(* CoDeSys 2.3 project: cy-08-wg-03.pro *)
(* Title: ClevergyAS - SanFelice *)
(* Version: 0.0 *)
(* Author: Andrea Ravasio *)
(* Libraries: serial_interface_01.lib 22.4.13 12:50:14, SerComm.lib 31.5.11 08:54:36, MBus_03.lib 9.2.13 17:51:58, Util.lib 18.5.10 15:14:28, Visual.lib 2.12.10 14:48:34, WagoLibIdent.lib 25.2.13 11:12:16, WagoLibStatus.lib 2.12.10 14:48:32, SysLibFile.lib 2.12.10 14:48:34, SysLibRtc.lib 2.12.10 14:48:32, SysLibSockets.lib 10.2.11 09:20:54, SysLibEvent.lib 2.12.10 14:48:34, SysLibPlcCtrl.lib 2.12.10 14:48:32, Standard.lib 2.12.10 14:48:34, SYSLIBCALLBACK.LIB 2.12.10 14:48:32, WagoLibModbus_IP_01.lib*24.7.13 15:05:58 *)

(* PLC configuration (modules and I/O channels)
0750-0402 4 DI 24 V DC 3.0ms [Type_1_4_Channels] node 0, in %IB0 out %QB0 {INTTypePAAssignment = PLC; INTTypeModule = plugged}
  AT %IX0.0 [BOOLOnX_I] Ch_1 Digital input
  AT %IX0.1 [BOOLOnX_I] Ch_2 Digital input
  AT %IX0.2 [BOOLOnX_I] Ch_3 Digital input
  AT %IX0.3 [BOOLOnX_I] Ch_4 Digital input
Fieldbus variables [FB_VARS] node 1, in %IB0 out %QB0
Flag variables [FLAG_VARS] node 2, in %IB0 out %QB0
Modbus-Master [MB_MASTER] node 3, in %IB0 out %QB0
*)

(* Global variable list: Global_Constants *)
VAR_GLOBAL CONSTANT

	Plant_SN			: DWORD :=8;   		(* S/N Impianto di telecontrollo *)
	Plant_SW_VER		: WORD  :=3;		(* Versione SW installata *)

	(* Parameters *)

	(* Filesystem *)
	FilesPath  			: STRING :='S:\';

	(* TCP Logger *)
	Logger_SERVER			: STRING:='';
	Logger_IP					: STRING:='178.33.227.41'; (*192.168.100.3'; (*' clevergyimpianti.it  *)*)
	Logger_PORT				: WORD  :=80;
	Logger_GETSTART		: STRING:='GET /cygmsrv/hsgm.ashx?';
	Logger_GETEND			: STRING:='$R$N$R$N';
	Logger_CHECK			: STRING:='True';
	Logger_CRLF				: STRING:='$R$N';
	Logger_DataFile			: STRING:='S:\LOG.DAT';
	Logger_DataFileOld		: STRING:='S:\LOG.BCK';
	Logger_IndexFile			: STRING:='S:\LOG.IDX';
	Logger_ConnRetries		: BYTE:=5;
	Logger_RecoverMsgs	: BYTE:=100;

	(* TCP Remote *)
	Remote_PORT			: WORD  :=44818;
	Remote_WELCOME		: STRING:='Connected$R$N';
	Remote_OK				: STRING:='OK$R$N';
	Remote_ERROR			: STRING:='ERROR$R$N';

	(* TCP Sockets *)
	MAX_SEND_TCP_SERVER					 : DWORD:=3000;(*60000*)
	MAX_RECEIVE_TCP_SERVER				 : DWORD:=3000;
	MAX_RECEIVE_TCP_SERVER_SOCKET	  : DWORD:=1500;
	MAX_SEND_TCP_CLIENT					 : DWORD:=3000;(*15000*)
	MAX_RECEIVE_TCP_CLIENT				 : DWORD:=1500;
	MAX_RECEIVE_TCP_CLIENT_SOCKET		 : DWORD:=1500;
	MAX_RECEIVE_UDP_SERVER				 : INT  :=1472;
	MAX_RECEIVE_UDP_CLIENT				 : INT  :=1472;
	CONNECT_WATCHDOG_TIME				 : TIME :=t#10s;

END_VAR

VAR_GLOBAL CONSTANT RETAIN
	TiemOutModbus_TCPIP				: TIME:=t#40ms;
	OffsetIndirizzo				: WORD := 0;(*12288;    (* questo servere per leggere il nodo WAGO *) *)

	MaxRigheFileCSV			:BYTE:=30; (* Massimo riche da leggere del afile csv *)
	MAXCaratteri				:WORD:=6000; (*Numero Massimo di caratteri da leggere dal file equivale alla lunghezza dei file*)


END_VAR

(* Global variable list: Global_Retain *)
VAR_GLOBAL RETAIN PERSISTENT
(*	CTL01_Count : DWORD;

	PortataTotalePORT01: DINT;
	ConteggioTotalePORT01: DINT;
	PortataTotaleGAS01: DINT;
	ConteggioTotaleGAS01: DINT;
	PortataTotaleGAS02: DINT;
	ConteggioTotaleGAS02: DINT;
*)
	Mode_Manual : BOOL := FALSE;
END_VAR

(* Global variable list: Global_Variables *)
VAR_GLOBAL

	SYS    : typ_SYS;


(* PLC *)

	Sistem_Status 							: INT ;
	BATTERY_STATUS 						: INT ;
	SYSTEM_STATUS_COMMAND 			: WORD;
	STATUS_DIGITAL_INPUT_1 				: WORD;
	STATUS_DIGITAL_OUTPUT_1			: WORD;
	STATUS_SYSTEM_WARNNG_1  			: WORD;
	STATUS_SYSTEM_ALARM_1 			: WORD;
	STATUS_SYSTEM_ALARM_2 			: WORD;

	PM1_Voltage_L12 						:REAL;
	PM1_Voltage_L23							:REAL;
	PM1_Voltage_L31 						:REAL;
	PM1_Current_L12						:REAL;
	PM1_Current_L23 						:REAL;
	PM1_Current_L31 						:REAL;
	PM1_Active_Power_Total 				:REAL;
	PM1_Reactive_Power_Total				:REAL;
	PM1_Apparent_Power_Total 				:REAL;
	PM1_Frequency 							:REAL;
	PM1_Power_Factor_Total 				:REAL;

(* GATEWAY BATTERY*)

	GW_Actual_DC_Voltage 					:REAL;
	GW_Actual_DC_Current 					:REAL;
	GW_Actual_Battery_SOC 				:REAL;
	GW_Actual_Heaters_Current 			:REAL;
	GW_Vdc_Link_Request 					:REAL;
	GW_Limit_Discharge_Current 			:REAL;
	GW_Limit_Charge_Current 				:REAL;
	GW_Min_DC_Voltage 					:REAL;
	GW_Max_DC_Voltage					:REAL;
	GW_Actual_Battery_Capacity 			:REAL;
	GW_Max_Battery_Voltage 				:REAL;
	GW_Min_Battery_Voltage 				:REAL;
	GW_Max_Battery_Temperature			:REAL;
	GW_Min_Battery_Temperature 			:REAL;
	GW_Actual_DC_Power 					:REAL;
	GW_HOURSOp_Time  					:INT;
	GW_MINOp_Time 						:INT;
	GW_Status_Warning_1 					:INT;
	GW_Status_Warning_2 					:INT;
	GW_Status_Alarm_1 						:INT;
	GW_Status_Alarm_2 						:INT;
	GW_Status_Warning_A 					:INT;
	GW_Status_Warning_B 					:INT;
	GW_Status_Alarm_A 						:INT;
	GW_CONTROLWORD  					:WORD ;
	GW_STATUSWORD  						:WORD;



(* PCS HPP 35*)

	PCS_Actual_Current_R 					 :REAL;
	PCS_Actual_Current_S 					 :REAL;
	PCS_Actual_Current_T 					 :REAL;
	PCS_Actual_Voltage_RS					 :REAL;
	PCS_Actual_Voltage_ST 					 :REAL;
	PCS_Actual_Voltage_TR					 :REAL;
	PCS_Frequency 							 :REAL;
	PCS_P_Actual 							 :REAL;
	PCS_Q_Actual 							 :REAL;
	PCS_A_Actual 							 :REAL;
	PCS_Battery_Voltage 						 :REAL;
	PCS_Battery_Current						 :REAL;
	PCS_Battery_Power 						 :REAL;
	PCS_PV_Voltage 							 :REAL;
	PCS_PV_Current 							 :REAL;
	PCS_PV_Power							 :REAL;
	PCS_HPP_Status 						 :INT;
	PCS_Drive_Status 						 :INT;
	PCS_Chopper_Status 					 :INT;
	PCS_Run_Mode 							 :INT;
	PCS_Drive_Warning_1  					 :WORD;
	PCS_Drive_Alarm_1  						 :WORD;
	PCS_HPP_Warning_1  					 :WORD;
	PCS_HPP_Alarm_1 						 :WORD ;


(* Write Register*)

	Ref_P										:REAL;

(* Variabile letta dal file CSV *)

	Ref_AvctivePower							:REAL;
	NomeFileSchedulazione					:STRING:='S:\Schedulazione.csv' ;
	WebStrutturaDati							: ARRAY [1..MaxRigheFileCSV] OF StrutturaDatiCSV;
	ForzaLetturaCSV: BOOL;

(* Variabile lettura ModBus ETH *)

	BitConnessione: BOOL ;    (* Abilita Comunicazione ModBus TCP-IP *)
	StartComunicazione: BOOL;
	ForzaLettura: BOOL;


	Logger : typ_Logger;

	(**** SIMULATION ONLY ****)
	TEST1		:BOOL;
	TEST2		:BOOL;

	T_S1		:INT:=100;

END_VAR


VAR_GLOBAL CONSTANT

END_VAR

(* Data type in Errors *)
TYPE en_Logger_ErrLev :
(
	EL_Log			:=0,
	EL_Wrn			:=1,
	EL_Alarm		:=2,
	EL_AlarmStop	:=3
);
END_TYPE

(* Data type in Errors *)
TYPE en_Logger_Status :
(
	S_Logger_UNKNOWN := 0,
	S_Logger_IDLE,
	S_Logger_WAITCONN,
	S_Logger_WAITTX,
	S_Logger_WAITRESP,
	S_Logger_ERROR
);
END_TYPE

(* Data type *)
TYPE en_SYS_Objects :
(
	EO_SYS		:=0,  (* PLC *)
	EO_VPN		:=1,  (* VPN *)
	EO_DOOR		:=2,  (* Door & access control *)

	EO_CAL		:=10, (* Caldaia *)
	EO_CIR		:=11, (* Circolatore *)
	EO_CRON		:=12, (* Crono-termostato *)
	EO_VRD		:=13, (* Valvola miscelatore pannelli *)
	EO_CTL		:=14, (* Contalitri *)
	EO_CTB		:=15, (* Contabilizzatore *)
	EO_TPV		:=16, (* Temperature probes & values *)
	EO_PPV		:=17, (* Pressure probes & values *)
	EO_PBV		:=18, (* Over-Pressure Alarms *)
	EO_TBV		:=19, (* Over-Temperature Alarms *)
	EO_PMV		:=20, (* Under-Pressure Alarms *)
	EO_GRU		:=21, (* Gruppo termico *)
	EO_PDC		:=22, (* Pompa di calore *)
	EO_SOL		:=23, (* Pannello solare termico *)
	EO_ESOL		:=24, (* Pannello solare fotovoltaico *)
	EO_GAS		:=25, (* Contatore GAS *)
	EO_PORT		:=26, (* Misuratore di portata *)

	EO_LON		:=1000, (* Bus - LON *)
	EO_MODBUS	:=1001, (* Bus - MODBUS *)
	EO_MBUS		:=1002  (* Bus - M-BUS *)
);
END_TYPE

(* Data type *)
TYPE en_SYS_Status :
(
	S_UNKNOWN  := 0,
	S_STARTUP,
	S_INIT_RTC,
	S_INIT_VAR,
	S_AUTOTEST,
	S_RUNNING,
	S_SHUTDOWN,
	S_HALT
);
END_TYPE

(* Data type in Plant_Objects *)
TYPE StrutturaDatiCSV :

STRUCT

	sdIndice: STRING(3);
	sdData: STRING(12);
	sdOra: STRING(6);
	sdOrigine: STRING(12);
	sdVaribile: STRING(10);
	sdValore: STRING(10);
END_STRUCT
END_TYPE

(* Data type in Plant_Objects *)
TYPE Typ_CTB_MBUS :
STRUCT
	Value			: STRING[21];
	Pof10			: STRING[3];
	Unit			: STRING[7];
	Descriptor		: STRING[6];
	(*Enum_Unit	: typMBusUnit; *)
END_STRUCT
END_TYPE

(* Data type in Errors *)
TYPE typ_Logger :
STRUCT
	Status		: en_Logger_Status;

	SendReq		: BOOL;
	SendIdx		: DWORD;
	SendData	: ARRAY [0..MAX_SEND_TCP_CLIENT] OF BYTE;
	SendLen		: DINT;

	TData		: ARRAY [0..MAX_SEND_TCP_CLIENT] OF BYTE;
	TLen		: DINT;

	LastIdxPos	: DWORD;

END_STRUCT
END_TYPE

(* Data type *)
TYPE typ_SYS :
STRUCT
	Status			: en_SYS_Status;
	Warning			: BOOL;
	Alarm			: BOOL;
	AlarmStop		: BOOL;

	Time_LogString	: STRING;
	Time_Year		: WORD;
	Time_Month		: BYTE;
	Time_Day		: BYTE;

	Time_CT_DT		: DT;
	Time_CT_Day		: WORD;
	Time_CT_Quarter	: BYTE;

	LastLogs_Idx	: BYTE;
	LastLogs_Dat	: ARRAY[0..5] OF STRING;
	LastLogs_Msg	: ARRAY[0..5] OF STRING;

END_STRUCT
END_TYPE

(* Data type in Plant_Objects *)
TYPE typ_VisuStrutturaMbus :
STRUCT

	sdNodoPresente: STRING(16);
	sdEnergia: STRING(16);
	sdPotenza: STRING(16);
	sdVolume: STRING(16);
	sdFlow: STRING(16);
	sdTempIngresso: STRING(8);
	sdTempaUscita: STRING(8);
	sdTempDelta: STRING(8);

END_STRUCT
END_TYPE

(* POU PLC_PRG, ST *)
PROGRAM PLC_PRG
VAR
	Timer1: TON; (* Fast controls tick *)
	Timer2: TON; (* Plant control tick *)
	Timer3: TON; (* Logger timer *)
	Timer4: TON; (* Logger timer *)
END_VAR
(******************************************************************************
 ****                           MAIN TASK CODE                             ****
 ******************************************************************************

	Network setup:
		IP  = 10.186.73.101 | MSK = 255.255.255.0 | GW = 10.186.73.254 
		DNS = ___.___.___.___ | NTP = ___.___.___.___

	Editor setup:
		Project --> Options --> Editor --> Fonts --> Courier NEW / BOLD / 12

*)

(*==============================*)
(*===== Main status machine ====*)
(*==============================*)
Main_Stm();
SceltaWrite();
(*=====================================*)
(*== Running common cycle operations ==*)
(*=====================================*)

IF SYS.Status>S_INIT_VAR THEN

(*	(* Execute M-BUS processes *)
	MBUS01();
	CTBSCAN01( MBus:=MBUS01.MBus ); *)

	ModBus_TCPIP();



END_IF

(*==============================*)
(*== System cycle operations ===*)
(*==============================*)
(* Execute TCP processes *)
Logger_Proc();
Remote_Proc();
(* Update user led *)
USRLED_Update();
(* Execute Cron Editor commands *)
(*...*)
(* External resources *)
(*...*)

(**** SIMULATION ONLY ****)
(*...*)
END_PROGRAM
ACTION Main_Stm:
CASE Sys.Status OF

	S_STARTUP:
		Sys.Status:=S_INIT_RTC;
		BitConnessione:=FALSE;

	S_INIT_RTC:
		(* Check RTC and update from network *)
		RTC_Update();
		(* Check time *)
		IF Sys.Time_Year>2000 THEN
			Sys.Status:=S_INIT_VAR;
		END_IF

	S_INIT_VAR:
		LogEv(EL_Wrn,EO_SYS,0,1,CONCAT('System_startup_v',WORD_TO_STRING(Plant_SW_VER)));
		Sys.Status:=S_RUNNING;
		BitConnessione:=TRUE;
		PRG_ApriFile( NomeFile:=NomeFileSchedulazione  ,  LungRecord:=4 );

	S_RUNNING:

		Timer1(IN:=NOT Timer1.Q,PT:=T#50ms);
(*		IF Timer1.Q THEN
			(* Update system checks *)
			(*SYS_Proc();*)
		END_IF
*)

		Timer2(IN:=NOT Timer2.Q AND NOT ForzaLettura ,PT:=T#10s); (* Lettura Variabili PLC Siemens via TCP-IP *)
		IF Timer2.Q OR ForzaLettura THEN
			(* Read current date/time *)
			RTC_Update();
			(* === Execute plant operations === *)
			StartComunicazione:=TRUE;
			(* Test toggle *)
			IF TEST1 THEN TEST1:=FALSE; ELSE TEST1:=TRUE; END_IF
		     END_IF

		Timer3(IN:=NOT Timer3.Q,PT:=T#5m);
		IF Timer3.Q THEN
			(* Trig logger *)
			LogTrig();
			(* Execute temporary CSV logger *)
(*			CSV_Log(); *)
		END_IF

		Timer4(IN:=NOT Timer4.Q AND NOT ForzaLetturaCSV,PT:=T#5m);    (* Lettura File Struttura *)
		IF Timer4.Q OR ForzaLetturaCSV THEN
			PRG_ApriFile( NomeFile:=NomeFileSchedulazione  ,  LungRecord:=4 );
		END_IF





	S_SHUTDOWN:
		(* Arresto del sistema *)
		Sys.Status:=S_STARTUP;
		BitConnessione:=FALSE;
	S_HALT:
		(* Aspetta uscita manuale *)
		Sys.Status:=S_STARTUP;


ELSE
	Sys.Status:=S_STARTUP;
END_CASE;
END_ACTION

(* POU Utils/SceltaWrite, ST *)
PROGRAM SceltaWrite
VAR
	TS: STRING;
	ORAttuale: INT;

	x: INT;
	OraImpostata: INT;
	StringaAggiornata: BOOL;
	Ref_AvctivePowerold: REAL;
END_VAR
(* scelgo la varibile da scrivere in funzione del'ora *)




(* Calculate variables *)
TS:=DT_TO_STRING(Sys.Time_CT_DT);
ORAttuale:=STRING_TO_INT(MID(STR:=TS, LEN:=2, POS:=15));


FOR x:=1 TO PRG_ApriFile.Riga BY 1 DO
       OraImpostata :=STRING_TO_INT(LEFT(WebStrutturaDati[x].sdOra,2));
	IF ORAttuale>=OraImpostata THEN
		Ref_AvctivePower:=STRING_TO_REAL((WebStrutturaDati[x].sdValore ));
		END_IF
END_FOR

IF Ref_AvctivePower <>  Ref_AvctivePowerold THEN
		 LogEv(EL_Log,0,3,1,'Reference_active_power_Aggiornato');    (*********************************** moreno **********************)
		 Ref_AvctivePowerold:=Ref_AvctivePower;
END_IF
END_PROGRAM

(* POU Utils/PRG_ApriFile, ST *)
PROGRAM PRG_ApriFile


VAR
	(* Varibili per l'apertura del del File CVS *)
	xStart:							BOOL;

	FileIdent: 						DWORD;
	CarattereLetto:				ARRAY[0..50000] OF BYTE;
	filesizev: 						DINT;
(*	RecordLetto: 					STRING(80); *)
	PrimoCarattereRiga: 			INT;
	NumCaratteri:					DINT;
	Record: 						INT;
	Carattere: 						STRING(1);

	Riga: INT;
(*	x: DWORD;*)

	StringaAppoggio: STRING;
	Valore2: REAL;

(*	BufferLetto:			ARRAY[0..186] OF BYTE; *)


	NumeroRighe: BOOL;
(*	bCarattere: BYTE; *)
	AggiornaDato: BOOL;

END_VAR

VAR_INPUT
	NomeFile:STRING(20);
	LungRecord: BYTE;
END_VAR
(* cerco il file se presente quindi dò l'OK*)


	FileIdent:=SysFileOpen(FileName:=NomeFile , Mode:='r');
	IF fileident<>0 THEN
		SysFileRead(File:=Fileident, Buffer:=ADR(CarattereLetto), Size:=SIZEOF(CarattereLetto));
		filesizev:=SysFileGetSize(FileName:=NomeFile);
		NumeroRighe:=SysFileEOF(FileIdent);
		IF filesizev>MAXCaratteri THEN
			filesizev:=MAXCaratteri;
		END_IF
		SysFileClose(File:=fileident);(*this function is blocking*)
		xStart:=TRUE;
	ELSE
		xStart:=FALSE;
		LogEv(EL_Alarm,0,3,1,'Errore_File_CSV_Non_Letto');    (*********************************** moreno **********************)

		RETURN;(*no such file available*)
	END_IF

IF xStart=TRUE THEN



	PrimoCarattereRiga:=0;
	NumCaratteri:=0;
	Record:=1;
	Riga:=1;
	StringaAppoggio:='';

(* Costruisco la stringa *)

		FOR NumCaratteri:=0 TO filesizev DO

					(* elimino i caratteri che non mi servono *)

					WHILE  CarattereLetto[NumCaratteri]=10 OR (*Caratterre ? *)
						(*	 CarattereLetto[NumCaratteri]=32 OR (*Caratterre   *) *)
							 CarattereLetto[NumCaratteri]=34 OR (*Caratterre " *)
							 CarattereLetto[NumCaratteri]=36 OR (*Caratterre ' *)
							 CarattereLetto[NumCaratteri]=39 DO
 							NumCaratteri:=NumCaratteri+1;
					END_WHILE


					(* Gestione Caratteri di controllo *)
					IF CarattereLetto[NumCaratteri]=13 THEN  (*Caratterre fine Riga  *)
						AggiornaDato:=TRUE;
					 END_IF
					IF CarattereLetto[NumCaratteri]=59 THEN (*Caratterre Separatore Record*)
						AggiornaDato:=TRUE;
					 END_IF

			IF aggiornaDato THEN

					(*Creo l'array nel PLC dei valori letti dal file  *)
				CASE Record OF

						1:	WebStrutturaDati[Riga].sdIndice:=INT_TO_STRING(RIGA);
							WebStrutturaDati[Riga].sdData:=LEFT(StringaAppoggio,10);
							WebStrutturaDati[Riga].sdOra:=RIGHT(StringaAppoggio,5);
							Record:=Record+1;
						2: 	WebStrutturaDati[Riga].sdOrigine:=StringaAppoggio;
							Record:=Record+1;
						3: 	WebStrutturaDati[Riga].sdVaribile:=StringaAppoggio;
							Record:=Record+1;
						4: 	WebStrutturaDati[Riga].sdValore:=StringaAppoggio;
							Record:=Record+1;

				END_CASE
				AggiornaDato:=FALSE;
				StringaAppoggio:='';
				IF Record>LungRecord THEN
						Record:=1;
						Riga:=Riga+1;
				 END_IF



			ELSE
					Carattere:=FUN_ByteAsci(CarattereLetto[NumCaratteri]);
					StringaAppoggio:=CONCAT(StringaAppoggio,Carattere);
			END_IF
		END_FOR

END_IF
END_PROGRAM

(* POU TCP_Logger/LogEv, ST *)
FUNCTION LogEv : BOOL
VAR_INPUT
	Level	: en_Logger_ErrLev;
	Object  : en_SYS_Objects;
	Index	: WORD;
	Error	: WORD;
	Message : STRING;
END_VAR
VAR
	s1 : STRING(160);
	i  : INT;
END_VAR
(* Execute error level operations *)
CASE Level OF
	EL_Wrn: 	Sys.Warning:=TRUE;
	EL_Alarm: 		Sys.Alarm:=TRUE;
	EL_AlarmStop: 	Sys.Alarm:=TRUE; (* GO TO STOP STATE!! *)
END_CASE

(* Fill lastlog list *)
s1:=CONCAT(Sys.Time_LogString,';Lev=');
s1:=CONCAT(s1,INT_TO_STRING(Level));
s1:=CONCAT(s1,';Obj=');
s1:=CONCAT(s1,INT_TO_STRING(Object));
s1:=CONCAT(s1,';Idx=');
s1:=CONCAT(s1,WORD_TO_STRING(Index));
s1:=CONCAT(s1,';Err=');
s1:=CONCAT(s1,WORD_TO_STRING(Error));
Sys.LastLogs_Dat[Sys.LastLogs_Idx]:=s1;
Sys.LastLogs_Msg[Sys.LastLogs_Idx]:=Message;
Sys.LastLogs_Idx:=Sys.LastLogs_Idx+1;
IF Sys.LastLogs_Idx>5 THEN Sys.LastLogs_Idx:=0; END_IF

(*---------------------------------------------------------------*)
(*---------------------------------------------------------------*)
Logger.TLen:=0;
(* Set GET header *)
ADDSTRING(ADR(Logger.TData), ADR(Logger_GETSTART), Logger.TLen);

(* Insert Header *)
s1:=INSERT('ID=&V=1&D=',DWORD_TO_STRING(Plant_SN),3);
s1:=CONCAT(s1,Sys.Time_LogString);
s1:=CONCAT(s1,'&S=');
IF Sys.Alarm THEN i:=2; ELSIF Sys.Warning THEN i:=1; ELSE i:=0; END_IF
s1:=CONCAT(s1,INT_TO_STRING(i));
ADDSTRING(ADR(Logger.TData), ADR(s1), Logger.TLen);

(* Insert ERR *)
s1:=CONCAT('&ERR=',INT_TO_STRING(Level));
s1:=CONCAT(s1,';');
s1:=CONCAT(s1,INT_TO_STRING(Object));
s1:=CONCAT(s1,';');
s1:=CONCAT(s1,WORD_TO_STRING(Index));
s1:=CONCAT(s1,';');
s1:=CONCAT(s1,WORD_TO_STRING(Error));
s1:=CONCAT(s1,';');
ADDSTRING(ADR(Logger.TData), ADR(s1), Logger.TLen);
s1:=Message;
ADDSTRING(ADR(Logger.TData), ADR(s1), Logger.TLen);

(* Finalize string *)
ADDSTRING(ADR(Logger.TData), ADR(Logger_GETEND), Logger.TLen);

(*---------------------------------------------------------------*)
(*---------------------------------------------------------------*)

Logger_Send();
END_FUNCTION

(* POU Utils Functions/ADDSTRING, ST *)
FUNCTION ADDSTRING : BOOL
VAR_INPUT
	pTxData: POINTER TO BYTE;
	pString: POINTER TO BYTE;
END_VAR
VAR_IN_OUT
	TxLen: DINT;
END_VAR
VAR
END_VAR
pTxData:=pTxData+TxLen;
WHILE pString^<>0 DO
	pTxData^:=pString^;
	pString:=pString+1;
	pTxData:=pTxData+1;
	TxLen:=TxLen+1;
END_WHILE
END_FUNCTION

(* POU TCP_Logger/Logger_Send, ST *)
FUNCTION Logger_Send : BOOL
VAR
	hFile: 	DWORD;
	pos:	DWORD;
END_VAR
(* Read log position *)
pos:=SysFileGetSize(Logger_DataFile);
(* Check log size, bckup and erase if no pending messages *)
IF pos>100000000 (*100M*) THEN
	hFile:=SysFileOpen(Logger_IndexFile,'r');
	IF hFile=0 THEN
		SysFileDelete(Logger_DataFileOld);
		SysFileRename(Logger_DataFile,Logger_DataFileOld);
		pos:=0;
	ELSE
		SysFileClose(hFile);
	END_IF
END_IF
(* Write message on log file *)
hFile:=SysFileOpen(Logger_DataFile,'a');
IF hFile<>0 THEN
	SysFileWrite(hFile, ADR(Logger.TData), Logger.TLen);
	SysFileClose(hFile);
ELSE
	Sys.Warning:=TRUE;
END_IF


(* Check logger status *)
IF Logger.SendReq=FALSE THEN
	(* Set log position for recovery *)
	Logger.SendIdx:=pos;
	(* Copy message data *)
	MEMCPY(ADR(Logger.TData),ADR(Logger.SendData),DINT_TO_WORD(Logger.TLen));
	Logger.SendLen:=Logger.TLen;
	(* Trigger request *)
	Logger.SendReq:=TRUE;
ELSE
	(* Add message position+size in recovery indexes *)
	hFile:=SysFileOpen(Logger_IndexFile,'a');
	SysFileWrite(hFile, ADR(pos), SIZEOF(pos));
	SysFileWrite(hFile, ADR(Logger.TLen), SIZEOF(Logger.TLen));
	SysFileClose(hFile);
END_IF
END_FUNCTION

(* POU Utils Functions/MEMCPY, ST *)
FUNCTION MEMCPY:BOOL
VAR_INPUT
	pSourceAddress:POINTER TO ARRAY[1..2] OF BYTE;
	pDestinationAddress:POINTER TO ARRAY[1..2] OF BYTE;
	BytesToCopy:WORD;
END_VAR
VAR
END_VAR
WHILE (BytesToCopy > 0) DO
	pDestinationAddress^[1]:=pSourceAddress^[1]; (* copy bytes from source to destination *)
	pDestinationAddress:=ADR(pDestinationAddress^[2]); (* increment destination *)
	pSourceAddress:=ADR(pSourceAddress^[2]);(* increment source *)
	BytesToCopy:=BytesToCopy -1; (* decrement number of bytes to copy *)
END_WHILE
END_FUNCTION

(* POU IMI/FUN/FUN_ByteAsci, ST *)
FUNCTION FUN_ByteAsci : STRING(1)
VAR_INPUT
	ByteIn:BYTE;
END_VAR
VAR
END_VAR
CASE ByteIn OF

	32: FUN_ByteAsci:=' ';
	33: FUN_ByteAsci:='!';
	34: FUN_ByteAsci:='"';
	35: FUN_ByteAsci:='#';

	37: FUN_ByteAsci:='%';
	38: FUN_ByteAsci:='&';

	40: FUN_ByteAsci:='(';
	41: FUN_ByteAsci:=')';
	42: FUN_ByteAsci:='*';
	43: FUN_ByteAsci:='+';
	44: FUN_ByteAsci:=',';
	45: FUN_ByteAsci:='-';
	46: FUN_ByteAsci:='.';
	47: FUN_ByteAsci:='/';
	48: FUN_ByteAsci:='0';
	49: FUN_ByteAsci:='1';
	50: FUN_ByteAsci:='2';
	51: FUN_ByteAsci:='3';
	52: FUN_ByteAsci:='4';
	53: FUN_ByteAsci:='5';
	54: FUN_ByteAsci:='6';
	55: FUN_ByteAsci:='7';
	56: FUN_ByteAsci:='8';
	57: FUN_ByteAsci:='9';
	58: FUN_ByteAsci:=':';
	59: FUN_ByteAsci:=';';
	60: FUN_ByteAsci:='<';
	61: FUN_ByteAsci:='=';
	62: FUN_ByteAsci:='>';
	63: FUN_ByteAsci:='?';
	64: FUN_ByteAsci:='@';
	65: FUN_ByteAsci:='A';
	66: FUN_ByteAsci:='B';
	67: FUN_ByteAsci:='C';
	68: FUN_ByteAsci:='D';
	69: FUN_ByteAsci:='E';
	70: FUN_ByteAsci:='F';
	71: FUN_ByteAsci:='G';
	72: FUN_ByteAsci:='H';
	73: FUN_ByteAsci:='I';
	74: FUN_ByteAsci:='J';
	75: FUN_ByteAsci:='K';
	76: FUN_ByteAsci:='L';
	77: FUN_ByteAsci:='M';
	78: FUN_ByteAsci:='N';
	79: FUN_ByteAsci:='O';
	80: FUN_ByteAsci:='P';
	81: FUN_ByteAsci:='Q';
	82: FUN_ByteAsci:='R';
	83: FUN_ByteAsci:='S';
	84: FUN_ByteAsci:='T';
	85: FUN_ByteAsci:='U';
	86: FUN_ByteAsci:='V';
	87: FUN_ByteAsci:='W';
	88: FUN_ByteAsci:='X';
	89: FUN_ByteAsci:='Y';
	90: FUN_ByteAsci:='Z';
	91: FUN_ByteAsci:='[';
	92: FUN_ByteAsci:='\';
	93: FUN_ByteAsci:=']';
	94: FUN_ByteAsci:='^';
	95: FUN_ByteAsci:='_';
	96: FUN_ByteAsci:='`';
	97: FUN_ByteAsci:='a';
	98: FUN_ByteAsci:='b';
	99: FUN_ByteAsci:='c';
	100: FUN_ByteAsci:='d';
	101: FUN_ByteAsci:='e';
	102: FUN_ByteAsci:='f';
	103: FUN_ByteAsci:='g';
	104: FUN_ByteAsci:='h';
	105: FUN_ByteAsci:='i';
	106: FUN_ByteAsci:='j';
	107: FUN_ByteAsci:='k';
	108: FUN_ByteAsci:='l';
	109: FUN_ByteAsci:='m';
	110: FUN_ByteAsci:='n';
	111: FUN_ByteAsci:='o';
	112: FUN_ByteAsci:='p';
	113: FUN_ByteAsci:='q';
	114: FUN_ByteAsci:='r';
	115: FUN_ByteAsci:='s';
	116: FUN_ByteAsci:='t';
	117: FUN_ByteAsci:='u';
	118: FUN_ByteAsci:='v';
	119: FUN_ByteAsci:='w';
	120: FUN_ByteAsci:='x';
	121: FUN_ByteAsci:='y';
	122: FUN_ByteAsci:='z';
	123: FUN_ByteAsci:='{';
	124: FUN_ByteAsci:='|';
	125: FUN_ByteAsci:='}';
	126: FUN_ByteAsci:='~';

	167: FUN_ByteAsci:='°';
	176: FUN_ByteAsci:='°';


ELSE
	FUN_ByteAsci:='';

END_CASE
END_FUNCTION

(* POU Plant_Objects/ModBus_TCPIP, ST *)
PROGRAM ModBus_TCPIP
VAR


	ModBusTCP: ETHERNET_MODBUSMASTER_TCP;

	StartReadIndirizzo: WORD := 400;
	ReadDaLeggere: WORD :=122;

	DatiLetti  : ARRAY [0..250] OF WORD; (* Dati Letti  *)

	StartWriteIndirizzo: WORD := 0;
	WriteDaScrivere: WORD := 20;
	DatiDaScrivere : ARRAY [0..20] OF WORD; (* Dati da scrivere *)


	NodoCollegato: BOOL;
	ErroreComunicazione: WORD;
	IndirizzoNodo: STRING := '10.186.73.105';



	TrgiFStartComunicazione_1: F_TRIG;
	TrgiFStartComunicazione_2: F_TRIG;

	TrgiRStartComunicazione: R_TRIG;

	DW_Appoggio: DWORD;

	Log_Status		: BYTE;
	Vis_StatusColor : DWORD;

	TrigRNodoCollegato: R_TRIG;
	TrigFNodoCollegato: F_TRIG;

END_VAR
(* Sul fronte di salita del Star Comunicazione aggiorna la variabiel da scrivere *)

TrgiRStartComunicazione(CLK:=StartComunicazione , Q=> );

IF TrgiRStartComunicazione.Q THEN

	Ref_P	:=Ref_AvctivePower;
	DW_Appoggio:=ConversioneReal_DWord(Ref_P);

	DatiDaScrivere[10]:=WORD_OF_DWORD(DW_Appoggio, 0);
	DatiDaScrivere[11]:=WORD_OF_DWORD(DW_Appoggio, 1);

END_IF





ModBusTCP(
				xCONNECT:= BitConnessione,
				strIP_ADDRESS:=IndirizzoNodo ,
				(*  wPORT:= , di default 502 *)
				(*  bUNIT_ID:= ,di default 0 *)
				bFUNCTION_CODE:= 23, (*0x17:	read and write multiple register*)
				wREAD_ADDRESS:=StartReadIndirizzo + OffsetIndirizzo ,
				wREAD_QUANTITY:= ReadDaLeggere,
				ptREAD_DATA:=ADR(DatiLetti) ,
				wWRITE_ADDRESS:=StartWriteIndirizzo + OffsetIndirizzo ,
				wWRITE_QUANTITY:= WriteDaScrivere,
				ptSEND_DATA:=ADR(DatiDaScrivere) ,
				tTIME_OUT:=TiemOutModbus_TCPIP ,
				(* 	tCON_WATCHDOG:= ,		:TIME:=t#1s;  *)
				xSEND:= StartComunicazione,

				xIS_CONNECTED=> NodoCollegato ,
				wERROR=> ErroreComunicazione ,
				bRESPONSE_UNIT_ID=> );


IF ErroreComunicazione<>0 AND NOT ( Log_Status=0) THEN
	Log_Status:=2; Vis_StatusColor:=16#2020F0;
       LogEv(EL_AlarmStop,ErroreComunicazione,3,1,'Errore_Comunicazione ');    (*********************************** moreno **********************)
  ELSE
	Log_Status:=0; Vis_StatusColor:=16#20F020;
END_IF

TrigRNodoCollegato(CLK:=NodoCollegato , Q=> );
TrigFNodoCollegato(CLK:= NodoCollegato, Q=> );

IF TrigFNodoCollegato.Q  THEN
       LogEv(EL_AlarmStop,ErroreComunicazione,3,1,'Nodo_Non_Collegato');    (*********************************** moreno **********************)
 END_IF


IF TrigRNodoCollegato.Q  THEN
       LogEv(EL_Log,0,1,1,'Nodo_Collegato');    (*********************************** moreno **********************)
 END_IF




TrgiFStartComunicazione_1(CLK:=StartComunicazione, Q=> );

(* Quando il Bit StartComunicazione torna a zero significa che la comunicazione è terminata quindi rilevo i dati *)
(*ricordiamo che si parte ad interrogare l'indirizzo 400 quindi l'array che è dimensionato 0..250 si leggeranno i valori 400..600*)
IF TrgiFStartComunicazione_1.Q AND NodoCollegato AND ErroreComunicazione=0 AND StartReadIndirizzo=400 THEN

(* PLC *)

	Sistem_Status:=DatiLetti[0];
	BATTERY_STATUS :=DatiLetti[1];
	SYSTEM_STATUS_COMMAND :=DatiLetti[10];
	STATUS_DIGITAL_INPUT_1 :=DatiLetti[15];
	STATUS_DIGITAL_OUTPUT_1 :=DatiLetti[20];
	STATUS_SYSTEM_WARNNG_1 :=DatiLetti[25];
	STATUS_SYSTEM_ALARM_1  :=DatiLetti[30];
	STATUS_SYSTEM_ALARM_2  :=DatiLetti[31];


	DW_Appoggio:=DatiLetti[36]*65535+DatiLetti[35];
	PM1_Voltage_L12:=ConversioneDword_Real(DW_Appoggio);

	DW_Appoggio:=DatiLetti[38]*65535+DatiLetti[37];
	PM1_Voltage_L23:=ConversioneDword_Real(DW_Appoggio);

	DW_Appoggio:=DatiLetti[40]*65535+DatiLetti[39];
	PM1_Voltage_L31:=ConversioneDword_Real(DW_Appoggio);

	DW_Appoggio:=DatiLetti[42]*65535+DatiLetti[41];
	PM1_Current_L12:=ConversioneDword_Real(DW_Appoggio);

	DW_Appoggio:=DatiLetti[44]*65535+DatiLetti[43];
	PM1_Current_L23:=ConversioneDword_Real(DW_Appoggio);

	DW_Appoggio:=DatiLetti[46]*65535+DatiLetti[45];
	PM1_Current_L31:=ConversioneDword_Real(DW_Appoggio);

	DW_Appoggio:=DatiLetti[48]*65535+DatiLetti[47];
	PM1_Active_Power_Total:=ConversioneDword_Real(DW_Appoggio);

	DW_Appoggio:=DatiLetti[50]*65535+DatiLetti[49];
	PM1_Reactive_Power_Total:=ConversioneDword_Real(DW_Appoggio);

	DW_Appoggio:=DatiLetti[52]*65535+DatiLetti[51];
	PM1_Apparent_Power_Total:=ConversioneDword_Real(DW_Appoggio);

	DW_Appoggio:=DatiLetti[54]*65535+DatiLetti[53];
	PM1_Frequency:=ConversioneDword_Real(DW_Appoggio);

	DW_Appoggio:=DatiLetti[56]*65535+DatiLetti[55];
	PM1_Power_Factor_Total:=ConversioneDword_Real(DW_Appoggio);


(* GATEWAY BATTERY*)

	DW_Appoggio:=DatiLetti[70]*65535+DatiLetti[69];
	GW_Actual_DC_Voltage:=ConversioneDword_Real(DW_Appoggio);

	DW_Appoggio:=DatiLetti[72]*65535+DatiLetti[71];
	GW_Actual_DC_Current:=ConversioneDword_Real(DW_Appoggio);

	DW_Appoggio:=DatiLetti[74]*65535+DatiLetti[73];
	GW_Actual_Battery_SOC:=ConversioneDword_Real(DW_Appoggio);

	DW_Appoggio:=DatiLetti[76]*65535+DatiLetti[75];
	GW_Actual_Heaters_Current:=ConversioneDword_Real(DW_Appoggio);

	DW_Appoggio:=DatiLetti[78]*65535+DatiLetti[77];
	GW_Vdc_Link_Request:=ConversioneDword_Real(DW_Appoggio);

	DW_Appoggio:=DatiLetti[80]*65535+DatiLetti[79];
	GW_Limit_Discharge_Current:=ConversioneDword_Real(DW_Appoggio);

	DW_Appoggio:=DatiLetti[82]*65535+DatiLetti[81];
	GW_Limit_Charge_Current:=ConversioneDword_Real(DW_Appoggio);

	DW_Appoggio:=DatiLetti[84]*65535+DatiLetti[83];
	GW_Min_DC_Voltage:=ConversioneDword_Real(DW_Appoggio);

	DW_Appoggio:=DatiLetti[86]*65535+DatiLetti[85];
	GW_Max_DC_Voltage:=ConversioneDword_Real(DW_Appoggio);

	DW_Appoggio:=DatiLetti[88]*65535+DatiLetti[87];
	GW_Actual_Battery_Capacity:=ConversioneDword_Real(DW_Appoggio);

	DW_Appoggio:=DatiLetti[92]*65535+DatiLetti[91];
	GW_Max_Battery_Voltage:=ConversioneDword_Real(DW_Appoggio);

	DW_Appoggio:=DatiLetti[94]*65535+DatiLetti[93];
	GW_Min_Battery_Voltage:=ConversioneDword_Real(DW_Appoggio);

	DW_Appoggio:=DatiLetti[96]*65535+DatiLetti[95];
	GW_Max_Battery_Temperature:=ConversioneDword_Real(DW_Appoggio);

	DW_Appoggio:=DatiLetti[98]*65535+DatiLetti[97];
	GW_Min_Battery_Temperature:=ConversioneDword_Real(DW_Appoggio);

	DW_Appoggio:=DatiLetti[100]*65535+DatiLetti[99];
	GW_Actual_DC_Power:=ConversioneDword_Real(DW_Appoggio);


	GW_HOURSOp_Time :=DatiLetti[109];
	GW_MINOp_Time  :=DatiLetti[110];
	GW_Status_Warning_1  :=DatiLetti[111];
	GW_Status_Warning_2  :=DatiLetti[112];
	GW_Status_Alarm_1 :=DatiLetti[113];
	GW_Status_Alarm_2 :=DatiLetti[114];
	GW_Status_Warning_A  :=DatiLetti[115];
	GW_Status_Warning_B  :=DatiLetti[116];
	GW_Status_Alarm_A 	 :=DatiLetti[117];
	GW_CONTROLWORD  :=DatiLetti[119];
	GW_STATUSWORD :=DatiLetti[120];

	StartReadIndirizzo:=600;
	StartComunicazione:=TRUE;

END_IF




ModBusTCP(
				xCONNECT:= BitConnessione,
				strIP_ADDRESS:=IndirizzoNodo ,
				(*  wPORT:= , di default 502 *)
				(*  bUNIT_ID:= ,di default 0 *)
				bFUNCTION_CODE:= 23, (*0x17:	read and write multiple register*)
				wREAD_ADDRESS:=StartReadIndirizzo + OffsetIndirizzo ,
				wREAD_QUANTITY:= ReadDaLeggere,
				ptREAD_DATA:=ADR(DatiLetti) ,
				wWRITE_ADDRESS:=StartWriteIndirizzo + OffsetIndirizzo ,
				wWRITE_QUANTITY:= WriteDaScrivere,
				ptSEND_DATA:=ADR(DatiDaScrivere) ,
				tTIME_OUT:=TiemOutModbus_TCPIP ,
				(* 	tCON_WATCHDOG:= ,		:TIME:=t#1s;  *)
				xSEND:= StartComunicazione,

				xIS_CONNECTED=> NodoCollegato ,
				wERROR=> ErroreComunicazione ,
				bRESPONSE_UNIT_ID=> );


IF ErroreComunicazione<>0 AND NOT ( Log_Status=0) THEN
	Log_Status:=2; Vis_StatusColor:=16#2020F0;
       LogEv(EL_AlarmStop,ErroreComunicazione,3,1,'Errore_Comunicazione ');    (*********************************** moreno **********************)
  ELSE
	Log_Status:=0; Vis_StatusColor:=16#20F020;
END_IF

TrigRNodoCollegato(CLK:=NodoCollegato , Q=> );
TrigFNodoCollegato(CLK:= NodoCollegato, Q=> );

IF TrigFNodoCollegato.Q  THEN
       LogEv(EL_AlarmStop,0,3,1,'Nodo_Non_Collegato');    (*********************************** moreno **********************)
 END_IF

IF TrigRNodoCollegato.Q  THEN
       LogEv(EL_Log,0,1,1,'Nodo_Collegato');    (*********************************** moreno **********************)
 END_IF




TrgiFStartComunicazione_2(CLK:=StartComunicazione, Q=> );



IF TrgiFStartComunicazione_2.Q AND NodoCollegato AND ErroreComunicazione=0 AND StartReadIndirizzo=600 THEN

(* PCS HPP 35*)

	DW_Appoggio:=DatiLetti[02]*65535+DatiLetti[01];
	PCS_Actual_Current_R:=ConversioneDword_Real(DW_Appoggio);

	DW_Appoggio:=DatiLetti[04]*65535+DatiLetti[03];
	PCS_Actual_Current_S:=ConversioneDword_Real(DW_Appoggio);

	DW_Appoggio:=DatiLetti[06]*65535+DatiLetti[05];
	PCS_Actual_Current_T:=ConversioneDword_Real(DW_Appoggio);

	DW_Appoggio:=DatiLetti[08]*65535+DatiLetti[07];
	PCS_Actual_Voltage_RS:=ConversioneDword_Real(DW_Appoggio);

	DW_Appoggio:=DatiLetti[10]*65535+DatiLetti[09];
	PCS_Actual_Voltage_ST:=ConversioneDword_Real(DW_Appoggio);

	DW_Appoggio:=DatiLetti[12]*65535+DatiLetti[11];
	PCS_Actual_Voltage_TR:=ConversioneDword_Real(DW_Appoggio);

	DW_Appoggio:=DatiLetti[14]*65535+DatiLetti[13];
	PCS_Frequency:=ConversioneDword_Real(DW_Appoggio);

	DW_Appoggio:=DatiLetti[16]*65535+DatiLetti[15];
	PCS_P_Actual:=ConversioneDword_Real(DW_Appoggio);

	DW_Appoggio:=DatiLetti[18]*65535+DatiLetti[17];
	PCS_Q_Actual:=ConversioneDword_Real(DW_Appoggio);

	DW_Appoggio:=DatiLetti[20]*65535+DatiLetti[19];
	PCS_A_Actual:=ConversioneDword_Real(DW_Appoggio);

	DW_Appoggio:=DatiLetti[22]*65535+DatiLetti[21];
	PCS_Battery_Voltage:=ConversioneDword_Real(DW_Appoggio);

	DW_Appoggio:=DatiLetti[24]*65535+DatiLetti[223];
	PCS_Battery_Current:=ConversioneDword_Real(DW_Appoggio);

	DW_Appoggio:=DatiLetti[26]*65535+DatiLetti[25];
	PCS_Battery_Power:=ConversioneDword_Real(DW_Appoggio);

	DW_Appoggio:=DatiLetti[28]*65535+DatiLetti[27];
	PCS_PV_Voltage:=ConversioneDword_Real(DW_Appoggio);

	DW_Appoggio:=DatiLetti[30]*65535+DatiLetti[29];
	PCS_PV_Current:=ConversioneDword_Real(DW_Appoggio);

	DW_Appoggio:=DatiLetti[32]*65535+DatiLetti[31];
	PCS_PV_Power:=ConversioneDword_Real(DW_Appoggio);


	PCS_HPP_Status :=DatiLetti[33];
	PCS_Drive_Status  :=DatiLetti[34];
	PCS_Chopper_Status :=DatiLetti[35];
	PCS_Run_Mode 	 :=DatiLetti[36];
	PCS_Drive_Warning_1  :=DatiLetti[37];
	PCS_Drive_Alarm_1 :=DatiLetti[38];
	PCS_HPP_Warning_1   :=DatiLetti[39];
	PCS_HPP_Alarm_1  :=DatiLetti[40];

StartReadIndirizzo:=400;

END_IF
END_PROGRAM

(* POU IMI/FUN/ConversioneReal_DWord, ST *)
FUNCTION ConversioneReal_DWord : DWORD
VAR_INPUT
	VarIn : REAL;
END_VAR
VAR
	pt : POINTER TO DWORD;
END_VAR
pt := ADR(VarIn);
ConversioneReal_DWord := pt^;
END_FUNCTION

(* POU IMI/FUN/WORD_OF_DWORD, ST *)
FUNCTION WORD_OF_DWORD : WORD
VAR_INPUT
	in : DWORD;
	N : BYTE;
END_VAR


(*
version 1.2	30. oct. 2008
programmer 	hugo
tested by	oscat

this function extracts a single word from the nth position from right (right is lowest byte)
the lower word (starting with Bit0 from in) is selected with N=0.
*)
WORD_OF_DWORD := DWORD_TO_WORD(SHR(in,SHL(n,4)));

(* revision history
hm	17. jan 2007	rev 1.0
	original version

hm	2. jan 2008		rev 1.1
	improved performance

hm	30. oct. 2008	rev 1.2
	improved performance
*)
END_FUNCTION

(* POU IMI/FUN/ConversioneDword_Real, ST *)
FUNCTION ConversioneDword_Real : REAL
VAR_INPUT
	VarIN:DWORD;

END_VAR
VAR
	Segno:INT;
	Esponente:INT;
	Mantissa:DWORD;
	pt : POINTER TO REAL;
END_VAR
(*
(* Trovo il Segno *)
IF  VarIN AND 2147483648 THEN
	Segno:=1;
ELSE
	Segno:=-1
END_IF


(* Trovo l' Epsonente *)
IF Segno=1 THEN
	Esponente:=SHR(VarIN,23);
ELSE
	Esponente:=(SHR(VarIN,23) -256 ;
END_IF
*)
pt := ADR(VarIN);
ConversioneDword_Real := pt^;
END_FUNCTION

(* POU TCP_Logger/Logger_Proc, ST *)
PROGRAM Logger_Proc
VAR
	c1:         	TCPCLIENT;

	Open:	    	BOOL;
	IpAddr:			DWORD;
	InetAddr:		DWORD;
	Connected:  	BOOL;
	Error:      	DINT;
	TxTrig:     	BOOL;
	RxData:			ARRAY [0..MAX_RECEIVE_TCP_CLIENT] OF BYTE;
	RxLen:			DINT;

	Retry:			BYTE;	(* Counter for connection retries *)
	Recovered:		BYTE;	(* Counter for recovered unsent messages *)

	i:				DINT;
	pos:			DWORD;
	hFile:			DWORD;

END_VAR
(*=== State machine ===*)
CASE Logger.Status OF

	S_Logger_UNKNOWN:
		(* Startup *)
		Logger.SendReq:=FALSE;
		Open:=FALSE;
		Logger.Status:=S_Logger_IDLE;

	S_Logger_IDLE:
		(* Wait request *)
		IF Logger.SendReq THEN
			(* Resolve server name or use static IP *)
			IF LEN(Logger_SERVER)=0 THEN
				InetAddr:=SysSockInetAddr(Logger_IP);
			ELSE
				IpAddr:=SysSockGetHostByName(ADR(Logger_SERVER));
				DWORDSWAP(pIn:=ADR(IpAddr), pOut:=ADR(InetAddr));
			END_IF
			TxTrig:=FALSE;
			RxLen:=0;
			(* Open connection *)
			Open:=TRUE;
			Logger.Status:=S_Logger_WAITCONN;
		END_IF

	S_Logger_WAITCONN:
		(* Wait connection *)
		IF Connected THEN
			(* Send data *)
			TxTrig:=TRUE;
			Logger.Status:=S_Logger_WAITTX;
		END_IF
		IF Error>0 THEN
			Open:=FALSE;
			Logger.Status:=S_Logger_ERROR;
		END_IF

	S_Logger_WAITTX:
		(* Wait transmission *)
		IF NOT TxTrig THEN
			Logger.Status:=S_Logger_WAITRESP;
		END_IF
		IF Error>0 THEN
			Open:=FALSE;
			Logger.Status:=S_Logger_ERROR;
		END_IF

	S_Logger_WAITRESP:
		(* Wait response *)
		IF Connected=FALSE (* OR TIMEOUT!! *) THEN
			Open:=FALSE;
			(* Check response *)
			IF RxLen>=4 AND CHKSTRING(pString:=ADR(RxData), pPattern:=ADR(Logger_CHECK)) THEN
				Logger.SendReq:=FALSE;
				Retry:=0;
				(* Check unsent messages to flush *)
				IF Recovered<Logger_RecoverMsgs THEN
					MsgChk();
					IF Logger.SendReq=TRUE THEN
						Recovered:=Recovered+1;
					ELSE
						Recovered:=0;
					END_IF
				ELSE
					Recovered:=0;
				END_IF
				Logger.Status:=S_Logger_IDLE;
			ELSE
				Logger.Status:=S_Logger_ERROR;
			END_IF
		END_IF

	S_Logger_ERROR:
		(* Connection error or send failure *)
		Retry:=Retry+1;
		IF Retry>Logger_ConnRetries THEN
			(* Save message as unsent *)
			MsgSave();
			Logger.SendReq:=FALSE;
			Retry:=0;
		END_IF
		Logger.Status:=S_Logger_IDLE;

ELSE
	Logger.Status:=S_Logger_UNKNOWN;
END_CASE


(*=== Execute client lib ===*)
c1(
	xOpenConnection			:= Open,
	dwInetAddr 				:= InetAddr,
	wPortNumber				:= Logger_PORT,
	ptSendData				:= ADR(Logger.SendData),
	diSendCount				:= Logger.SendLen,
	tConnectWatchdogTime	:= t#10s,
	xStartSend				:= TxTrig,
	aReceiveBuffer			:= RxData,
	diReceiveCount			:= RxLen,
	xConnected				=> Connected,
	diError					=> Error
);

(*=== Process Rx data ===*)
(*IF RxLen>0 THEN
	RxLen:=0;
END_IF*)
END_PROGRAM
ACTION MsgChk:
(* Open index file *)
hFile:=SysFileOpen(Logger_IndexFile,'r');
IF hFile=0 THEN
	RETURN;
END_IF
(* Search oldest message to recover *)
SysFileSetPos(hFile,Logger.LastIdxPos);
Logger.SendLen:=0;
REPEAT
	SysFileRead(hFile, ADR(Logger.SendIdx), SIZEOF(Logger.SendIdx));
	pos:=SysFileGetPos(hFile);
	SysFileRead(hFile, ADR(Logger.SendLen), SIZEOF(Logger.SendLen));
UNTIL
	SysFileEOF(hFile) OR Logger.SendLen<>0
END_REPEAT
SysFileClose(hFile);
(* Delete index file when all messages are recovered *)
IF Logger.SendLen=0 THEN
	Logger.LastIdxPos:=0;
	SysFileDelete(Logger_IndexFile);
	RETURN;
END_IF
(* Recover message data *)
hFile:=SysFileOpen(Logger_DataFile,'r');
IF hFile<>0 THEN
	SysFileSetPos(hFile,Logger.SendIdx);
	SysFileRead(hFile,ADR(Logger.SendData),Logger.SendLen);
	Logger.SendReq:=TRUE;
	SysFileClose(hFile);
END_IF
(* Clear index entry *)
hFile:=SysFileOpen(Logger_IndexFile,'a');
IF hFile<>0 THEN
	SysFileSetPos(hFile,pos);
	i:=0;
	SysFileWrite(hFile, ADR(i), 4);
	Logger.LastIdxPos:=SysFileGetPos(hFile);
	SysFileClose(hFile);
END_IF
END_ACTION
ACTION MsgSave:
(* Add log position in recovery indexes *)
hFile:=SysFileOpen(Logger_IndexFile,'a');
SysFileWrite(hFile, ADR(Logger.SendIdx), SIZEOF(Logger.SendIdx));
SysFileWrite(hFile, ADR(Logger.SendLen), SIZEOF(Logger.SendLen));
SysFileClose(hFile);
END_ACTION

(* POU Utils Functions/TCPCLIENT, ST *)
FUNCTION_BLOCK TCPCLIENT
(***********************************************************************************************************	*)
(* Version: 1.3b                        			          													*)
(* Date: 28.10.2014                   				          							            			*)
(***********************************************************************************************************	*)
(* WAGO Kontakttechnik GmbH Hansastr. 27 32423 Minden(Westf.)													*)
(* Tel. +0049 571/887-0 Fax. +0049 571/887-0																	*)
(* Author: VB																									*)
(***********************************************************************************************************	*)
(*Description:	A TCP client to read and write data with additional connection watchdog							*)
(*History:																										*)
(*Version 1.3b: 28.10.2014: Use DWORD address for IP (Andrea Ravasio)											*)
(*Version 1.3: 11.02.2011: Changes according to 750-880/881											 			*)
(*Version 1.2: 29.08.2007 Bugfix TCP Client																		*)
(*Version 1.1: 15.01.2007 Changes according to FW11																*)
(*Version 1.0: 09.03.2006 Release																				*)
(***********************************************************************************************************	*)
VAR CONSTANT
	STATE_CREATE     				 : BYTE:= 0;
	STATE_OPEN     					 : BYTE:= 1;
	STATE_IOCTL    					 : BYTE:= 2;
	STATE_CONNECT     				 : BYTE:= 10;
	STATE_TX       					 : BYTE:= 20;
	STATE_RX       					 : BYTE:= 30;
	STATE_CLOSE    					 : BYTE:= 40;
	STATE_ERROR_TRAP			     : BYTE:= 200;
END_VAR

VAR_INPUT
	xOpenConnection					: BOOL;
	dwInetAddr						: DWORD; (* <== Use SysSockInetAddr() value or
													swapped bytes order of SysSockGetHostByName() value *)
	wPortNumber						: WORD;
	ptSendData						: POINTER TO ARRAY[0..MAX_SEND_TCP_CLIENT] OF BYTE;
	diSendCount						: DINT;
	tConnectWatchdogTime		    : TIME := t#10s;
END_VAR
VAR_OUTPUT
	xConnected						: BOOL;
	diError 						: DINT := 0;
END_VAR
(* ErrorCodes -----------------------------------------
	16#8001 => No socket descriptor available 
	16#8002 => SysSockSend returns -1 
	16#8003 => Socket was "gracefully closed" 
	16#8004 => switching to none blocking mode fails
	16#8005 => SysSockClose() returns FALSE 
    16#8006 => SysSockConnect() fails
    16#8007 => SysSockSend() fails
	16#8008 => error state machine 
	16#8009 => timeout while waiting for data from server 
------------------------------------------------------------*)
VAR_IN_OUT
	xStartSend							: BOOL;
	aReceiveBuffer						: ARRAY [0..MAX_RECEIVE_TCP_CLIENT] OF BYTE;
	diReceiveCount						: DINT;
END_VAR
VAR
	m_State								: BYTE := 0;
	m_ReceiveBuffer						: ARRAY [0..MAX_RECEIVE_TCP_CLIENT_SOCKET] OF BYTE;
	m_Socket							: DINT;
	m_AddressInfo						: SOCKADDRESS;
	m_BytesReceived						: DINT;
	m_diReturn							: DINT;
	m_xReturn							: BOOL;
	m_IoCtlParameter  					: DINT := 1; (* IOCTL-Parameter for non-blocking mode of sockets *)
	i									: INT;
	T_Connect							: TON;
	m_count								: DINT;
	diOption							: DINT := 1;
	m_Blocking   						: DINT := 0;
END_VAR
IF xOpenConnection THEN
	(* State maschine *)
	CASE  m_State OF

	(* -------------------------------------------------------------------------*)
	STATE_CREATE:
			(* create socket descriptor*)
			m_Socket := SysSockCreate(diAddressFamily	:= SOCKET_AF_INET,
													 diType		:= SOCKET_STREAM,
													 diProtocol := SOCKET_IPPROTO_TCP);
			IF m_Socket >= 0 THEN
			(*Set Push-Bit*)
				IF ADR(%MW0)=16#30000000  OR ADR(%MW0)=16#20000000 THEN (*841 or 881*)
					SysSockSetOption(
						diSocket:=m_Socket,
						diLevel:=6,
						diOption:=SOCKET_TCP_NODELAY,
						pOptionValue:=ADR(diOption),
						diOptionLength:=SIZEOF(diOption));
				ELSE
						;
				END_IF
				m_State := STATE_IOCTL; (* succesful *)
			ELSE
				diError := 16#8001;  (* no socket descriptor available *)
				m_State := STATE_ERROR_TRAP;
			END_IF

	(* -------------------------------------------------------------------------*)
	STATE_IOCTL: (* change  socket mode  to none blocking *)
		m_diReturn := SysSockIoctl( m_Socket, SOCKET_FIONBIO, ADR(m_IoCtlParameter));
		IF m_diReturn <> 0 THEN
			m_AddressInfo.sin_family := SOCKET_AF_INET;
			m_AddressInfo.sin_port := SysSockNtohs(wPortNumber);
			m_AddressInfo.sin_addr := dwInetAddr;
			m_State := STATE_CONNECT;
		ELSE
			diError := 16#8004;  (* switching to none blocking mode fails *)
			m_State := STATE_ERROR_TRAP;
		END_IF


	(* -------------------------------------------------------------------------*)
	STATE_CONNECT: (* connect with server *)
		T_Connect(IN:=TRUE , PT:=tConnectWatchdogTime);(*activate watchdog for establishing connection to a server*)
		m_xReturn := SysSockConnect ( m_Socket, ADR(m_AddressInfo),  SIZEOF(m_AddressInfo));
		IF m_xReturn THEN (* succesful *)
			IF xStartSend THEN
				m_State := STATE_TX;(*transmit data*)
			ELSE
				m_State := STATE_RX;(*wait for data from server*)
			END_IF
			xConnected:=TRUE;
			T_Connect(IN:=FALSE);
		ELSE
			IF T_Connect.Q THEN
				diError := 16#8006;  (* connect fails *)
				xConnected:=FALSE;
				T_Connect(IN:=FALSE);
				m_State := STATE_ERROR_TRAP;
				SysSockClose( m_Socket);
			ELSE
				m_State := STATE_CONNECT;(*client still  tries to set up connection*)
			END_IF
		END_IF


	STATE_TX:	 (* send TCP-message *)
		m_diReturn := SysSockSend(diSocket := m_Socket,
								  pbyBuffer := ADR(ptSendData^[0]),
								  diBufferSize := diSendCount-m_count,
								  diFlags := 0);

		CASE m_diReturn OF
		-1:	(* ERROR *)
			T_Connect(IN:=TRUE , PT:=CONNECT_WATCHDOG_TIME);(*activate watchdog to check communication*)
			IF t_Connect.Q THEN
				diError := 16#8007;
				T_Connect(IN:=FALSE);
				m_State:=STATE_CLOSE;
			END_IF
		0: (* socket was "gracefully closed" *)
			m_State := STATE_CLOSE;
			diError := 16#8003;
		ELSE (* succesful *)
			m_count:=m_count+m_diReturn;
			IF m_count>=diSendCount THEN
				diError := 16#0000;
				m_State := STATE_RX;
				m_count:=0;
				xStartSend:=FALSE;
			END_IF
			T_Connect(IN:=FALSE);
		END_CASE

	(* -------------------------------------------------------------------------*)
	STATE_RX: (* process receive data *)
			m_BytesReceived := SysSockRecv(	diSocket 	:= m_Socket,
										pbyBuffer 	:= ADR(m_ReceiveBuffer),		(* Address of receive buffer *)
										diBufferSize:= SIZEOF(m_ReceiveBuffer),
										diFlags		:= 0);

			CASE m_BytesReceived OF
			-1:	(* No data available or error occured *)
				T_Connect(IN:=TRUE , PT:=tConnectWatchdogTime);(*activate watchdog to check communication*)
				IF t_Connect.Q THEN
					diError:=16#8009;
					T_Connect(IN:=FALSE);
					m_State:=STATE_CLOSE;
				END_IF
				IF xStartSend THEN
					m_State:=STATE_TX	;(* WAIT IN THIS STATE  and check for arriving data or new send command*)
				END_IF;
			0: (* socket was "gracefully closed"  *)
				m_State:=STATE_CLOSE;
				diError := 16#8003;
			ELSE (* succesful *)
				diError := 16#0000;
				T_Connect(IN:=FALSE);
				(* Copy received data into receive buffer *)
				FOR i:= 0 TO DINT_TO_INT(m_BytesReceived	)-1 DO
					aReceiveBuffer[diReceiveCount]:= m_ReceiveBuffer[i];
					diReceiveCount:=(diReceiveCount+1) MOD SIZEOF(aReceiveBuffer);
				END_FOR

			END_CASE

	(* -------------------------------------------------------------------------*)
	STATE_CLOSE : (* close socket *)
		IF ADR(%MW0)=16#30000000  OR ADR(%MW0)=16#20000000 THEN (*841 or 881*)
			;
		ELSE
			SysSockShutdown(m_Socket, 0);;(*870*)
		END_IF
		m_xReturn := SysSockClose( m_Socket);
		m_Socket := -1;
		m_State := 0; (* succesful *)
		xConnected:=FALSE;
		T_Connect(IN:=FALSE);
	(* -------------------------------------------------------------------------*)
	STATE_ERROR_TRAP: (* error handling *)
		xConnected:=FALSE;

	ELSE  (* Bad FSM code trap  *)
			m_State:= STATE_ERROR_TRAP;
			diError:= 16#8008;
	END_CASE

ELSE(*close connection*)
	IF m_Socket >= 0 THEN
		IF ADR(%MW0)=16#30000000  OR ADR(%MW0)=16#20000000 THEN (*841 or 881*)
			;
		ELSE
			SysSockShutdown(m_Socket, 0);;(*870*)
		END_IF
		SysSockClose( m_Socket);
	END_IF
	m_Socket := -1;
	diError := 16#0000;
	m_State := STATE_CREATE;
	xConnected:=FALSE;
	T_Connect(IN:=FALSE);
END_IF
END_FUNCTION_BLOCK

(* POU Utils Functions/DWORDSWAP, ST *)
FUNCTION DWORDSWAP:BOOL
VAR_INPUT
	pIn:POINTER TO ARRAY[1..4] OF BYTE;
	pOut:POINTER TO ARRAY[1..4] OF BYTE;
END_VAR
VAR
END_VAR
pOut^[1]:=pIn^[4];
pOut^[2]:=pIn^[3];
pOut^[3]:=pIn^[2];
pOut^[4]:=pIn^[1];
END_FUNCTION

(* POU Utils Functions/CHKSTRING, ST *)
FUNCTION CHKSTRING : BOOL
VAR_INPUT
	pString: POINTER TO BYTE;
	pPattern: POINTER TO BYTE;
END_VAR
VAR
END_VAR
CHKSTRING:=TRUE;
WHILE pPattern^<>0 AND CHKSTRING DO
	IF pPattern^<>pString^ THEN CHKSTRING:=FALSE; END_IF
	pString:=pString+1;
	pPattern:=pPattern+1;
END_WHILE
END_FUNCTION

(* POU TCP_Remote/Remote_Proc, ST *)
PROGRAM Remote_Proc
VAR
	s1:         	TCPSERVER;
	Enable: 		BOOL;
	Connected: 		BOOL;
	Error: 			DINT;

	TxData:			ARRAY[0..MAX_SEND_TCP_SERVER] OF BYTE;
	TxLen:			DINT;
	TxTrig:			BOOL;

	RxData:			ARRAY [0..MAX_RECEIVE_TCP_SERVER] OF BYTE;
	RxLen:			DINT;

	Status:			DINT;

	(* Command interpreter *)

	Cmd_Buf:		ARRAY [0..MAX_RECEIVE_TCP_SERVER] OF BYTE;
	Cmd_Buf_U16:	POINTER TO WORD;
	Cmd_Buf_INT:	POINTER TO INT;
	Cmd_BufLen:		WORD;
	Cmd_St:			WORD;

	Cmd_Obj:		WORD;
	Cmd_ObjIdx:		WORD;
	Cmd_C:			WORD;
	Cmd_R:			WORD;
	Cmd_CLen:		WORD;
	Cmd_RLen:		WORD;

	i : WORD;
	j : INT;

END_VAR
(*=== State machine ===*)
CASE Status OF
	0: (* Startup *)
		TxLen:=0; TxTrig:=FALSE;
		RxLen:=0;
		Enable:=TRUE;
		Status:=1;

	1: (* Wait incoming connection *)
		IF Connected THEN
			(* Send welcome message *)
			ADDSTRING(pTxData:=ADR(TxData), pString:=ADR(Remote_WELCOME), TxLen:=TxLen);
			TxTrig:=TRUE;
			Cmd_BufLen:=0;
			Cmd_St:=0;
			Status:=2;
		END_IF
		IF Error>1 THEN
			Enable:=FALSE;
			Status:=0;
		END_IF

	2: (* Wait command *)
		IF RxLen>0 THEN
			(*=== Interpreter start ===*)
			IF Cmd_BufLen+(RxLen/2)>=MAX_RECEIVE_TCP_SERVER THEN
				(* ERROR *)
				Cmd_BufLen:=0;
			ELSE
				i:=HEXTORAW(pString:=ADR(RxData), StringLen:=DINT_TO_WORD(RxLen), pData:=ADR(Cmd_Buf[Cmd_BufLen]));
				Cmd_BufLen:=Cmd_BufLen+i;
			END_IF
			IF Cmd_BufLen>=8 THEN
				Cmd_Buf_U16:=ADR(Cmd_Buf[6]);
				IF Cmd_BufLen>=(8+Cmd_Buf_U16^) THEN
					Cmd_CLen:=Cmd_Buf_U16^;
					Cmd_Buf_U16:=ADR(Cmd_Buf[0]); Cmd_Obj:=Cmd_Buf_U16^;
					Cmd_Buf_U16:=ADR(Cmd_Buf[2]); Cmd_ObjIdx:=Cmd_Buf_U16^;
					Cmd_Buf_U16:=ADR(Cmd_Buf[4]); Cmd_C:=Cmd_Buf_U16^;
					Command();
					Cmd_BufLen:=0;
				END_IF
			END_IF

			(*=== Interpreter end ===*)
			RxLen:=0;
		END_IF
		IF NOT Connected THEN
			Status:=1;
		END_IF

ELSE
	Status:=0;
END_CASE


(*=== Execute server lib ===*)
s1(
	xEnable				:= Enable,
	wPortNumber			:= Remote_PORT,
	tServerTimeOut		:= t#15m,
	ptSendData			:= ADR(TxData),
	diSendCount			:= TxLen,
	xStartSend			:= TxTrig,
	aReceiveBuffer		:= RxData,
	diReceiveCount		:= RxLen,
	xClientConnected	=> Connected,
	diError				=> Error
);
END_PROGRAM
ACTION Cmd_CTB:
(* Check index *)
IF Cmd_ObjIdx<>1 THEN
	Cmd_R:=2;
	RETURN;
END_IF

(*
(* Process command *)
CASE Cmd_C OF

	1: (* START SCANNING *)
(*	CTBSCAN01.Refresh:=TRUE *)
		1:=1;
ELSE
	Cmd_R:=3;
END_CASE
*)
Cmd_R:=3;
END_ACTION
ACTION Cmd_SYS:
(* Check index *)
IF Cmd_ObjIdx<>0 THEN
	Cmd_R:=2;
	RETURN;
END_IF

(* Process command *)
CASE Cmd_C OF

	0: (* ECHO *)
		IF Cmd_CLen<>0 THEN
			TxLen:=0;
		END_IF

	1: (* LOG REQUEST *)
		LogTrig();

	2: (* REARM *)
		Sys.Warning:=FALSE;
		Sys.Alarm:=FALSE;
		Sys.AlarmStop:=FALSE;

ELSE
	Cmd_R:=3;
END_CASE
END_ACTION
ACTION Command:
(* Default response OK/NODATA *)
Cmd_R:=0;
Cmd_RLen:=0;
TxLen:=16;

(* Check object *)
CASE Cmd_Obj OF

	EO_SYS:
		Cmd_SYS();

ELSE
	Cmd_R:=1;
END_CASE

(* Generate response *)
IF TxLen>0 THEN
	RAWTOHEX(ADR(Cmd_Obj)	,2,ADR(TxData[ 0]));
	RAWTOHEX(ADR(Cmd_ObjIdx),2,ADR(TxData[ 4]));
	RAWTOHEX(ADR(Cmd_R)		,2,ADR(TxData[ 8]));
	RAWTOHEX(ADR(Cmd_RLen)	,2,ADR(TxData[12]));
	TxTrig:=TRUE;
END_IF
END_ACTION

(* POU Utils Functions/TCPSERVER, ST *)
FUNCTION_BLOCK TCPSERVER
(***********************************************************************************************************	*)
(* Version: 1.6                                    			          											*)
(* Date: 11.02.2011                                   					          							    *)
(***********************************************************************************************************	*)
(* WAGO Kontakttechnik GmbH Hansastr. 27 32423 Minden(Westf.)													*)
(* Tel. +0049 571/887-0 Fax. +0049 571/887-0																	*)
(* Author: VB																									*)
(***********************************************************************************************************	*)
(*Description:	A TCP server to read and write data													       		*)
(*Historie:																										*)
(*Version 1.6: 11.02.2011: Changes according to 750-880/881											 			*)
(*Version 1.5: 27.11.2008 Bugfix allow reuse port																*)
(*Version 1.4: 13.10.2008 Bugfix transmitting large data														*)
(*Version 1.3: 15.01.2007 Changes according to FW11																*)
(*Version 1.2: 09.03.2006 Changes for socket handle 0											       			*)
(*Version 1.1: 14.02.2005 Release																				*)
(***********************************************************************************************************	*)
VAR CONSTANT
	STATE_INIT     				 : BYTE:= 0;
	STATE_OPEN     				 : BYTE:= 1;
	STATE_TX       				 : BYTE:= 20;
	STATE_RX       				 : BYTE:= 30;
	STATE_CLOSE    				 : BYTE:= 40;
	STATE_ERROR_TRAP		 	 : BYTE:= 200;
END_VAR
VAR_INPUT
	xEnable    					: BOOL;	 (* Set TRUE to enable function block *)
	wPortNumber					: WORD;  (* Port *)
	tServerTimeOut				: TIME:=t#50s;
	ptSendData					: POINTER TO ARRAY[0..MAX_SEND_TCP_SERVER] OF BYTE;
	diSendCount					: DINT;
END_VAR
VAR_OUTPUT
	xClientConnected  			: BOOL:= FALSE;
	diError 					: DINT:= 0;
END_VAR
(* Status Codes -----------------------------------------
	16#8001 => No socket descriptor available 
	16#8002 => SysSockBind fails 
	16#8003 => SysSockListen fails 
	16#8004 => switching to none blocking mode fails
	16#8005 => SysSockClose() returns FALSE 
    16#8006 => SysSockConnect() fails
    16#8007 => SysSockSend() fails
	16#8008 => error state machine 
	16#8009 => timeout while waiting for data from server 
	16#0001 => server waiting for client to establish connection
------------------------------------------------------------*)
VAR_IN_OUT
	xStartSend					: BOOL;
	aReceiveBuffer				: ARRAY [0..MAX_RECEIVE_TCP_SERVER] OF BYTE;
	diReceiveCount				: DINT;
END_VAR

VAR
	m_State    					: BYTE:= 0;
	m_ReceiveBuffer				: ARRAY [0..MAX_RECEIVE_TCP_SERVER_SOCKET] OF BYTE;
	m_ServerSocket				: DINT:= SOCKET_INVALID;
	m_Socket					: DINT:= SOCKET_INVALID;
	m_AddressInfo				: SOCKADDRESS;
	m_BytesReceived				: DINT;
	m_diReturn					: DINT;
	m_xReturn					: BOOL;
	m_SizeSockadr				: DWORD;
	m_ConnectionWatchdog		: TON;
	m_Flags						: DINT;
	m_NoneBlocking   			: DINT:= 1;
	m_Blocking   				: DINT:= 0;
	i							: INT;
	m_count						: DINT;
	diOption					: DINT := 1;
	on: DINT;
END_VAR
IF xEnable THEN
	CASE m_State OF
		STATE_INIT:
			(* Create Socket *)
			m_ServerSocket:= SysSockCreate( SOCKET_AF_INET, SOCKET_STREAM, 0);
			IF m_ServerSocket = SOCKET_INVALID THEN
				(* *)
				diError:= 16#8001;
				m_State:= STATE_ERROR_TRAP;
				RETURN;
			ELSE
				;
			END_IF
			(* Address bindings *)
			(********************)
			on:=1;
			SysSockSetOption( m_ServerSocket, SOCKET_SOL, SOCKET_SO_REUSEADDR, ADR(on), SIZEOF(on) );

			m_AddressInfo.sin_family:= SOCKET_AF_INET;
			m_AddressInfo.sin_port  := SysSockHtons( wPortNumber);
			m_AddressInfo.sin_addr  := SOCKET_INADDR_ANY;
			IF NOT SysSockBind( m_ServerSocket, ADR(m_AddressInfo), SIZEOF(m_AddressInfo)) THEN
				diError:= 16#8002;
				m_State:= STATE_ERROR_TRAP;
				RETURN;
			END_IF
			(* Wait for connections *)
			(************************)
			IF NOT SysSockListen( m_ServerSocket, 1) THEN
				diError:= 16#8003;
				m_State:= STATE_ERROR_TRAP;
			END_IF

			(* Puts SOCKET in NonBlocking mode *)
			m_diReturn:= SysSockIoctl( m_ServerSocket, SOCKET_FIONBIO, ADR(m_NoneBlocking));

			m_State:= STATE_OPEN;


		STATE_OPEN: 	(* Waiting for incomming connection *)
				m_SizeSockadr:=SIZEOF(m_AddressInfo);
				m_Socket:= SysSockAccept( m_ServerSocket, ADR(m_AddressInfo), ADR(m_SizeSockadr));
				diError:=State_open;
				IF m_Socket <> SOCKET_INVALID THEN
					xClientConnected:=TRUE;
					(*Set Push-Bit:new V1.5*)
					IF ADR(%MW0)=16#30000000  OR ADR(%MW0)=16#20000000 THEN (*841 or 881*)
						SysSockSetOption(
							diSocket:=m_Socket,
							diLevel:=6,
							diOption:=SOCKET_TCP_NODELAY,
							pOptionValue:=ADR(diOption),
							diOptionLength:=SIZEOF(diOption));
					ELSE
							;
					END_IF
					SysSockIoctl( m_Socket, SOCKET_FIONBIO, ADR(m_NoneBlocking));
					m_State:= STATE_RX;
					diError:=0;
				END_IF

		STATE_RX:
					m_BytesReceived:= SysSockRecv( m_Socket, ADR(m_ReceiveBuffer), SIZEOF(m_ReceiveBuffer), 0);
					CASE m_BytesReceived OF
					-1:(*no data available or error occured*)
						m_ConnectionWatchdog(IN:=TRUE , PT:=tServerTimeOut );
						IF m_connectionWatchdog.Q THEN
							m_State:= STATE_CLOSE;
							m_ConnectionWatchdog(IN:=FALSE);(*reset connection watchdog*)
							diError := 16#8009;
						END_IF
					0:(* socket was "gracefully closed"  *)
						m_State:= STATE_CLOSE;
						diError := 16#8003;
					ELSE
						(* Copy received data into receive buffer *)
						(********************************)
						FOR i:= 0 TO DINT_TO_INT(m_BytesReceived	)-1 DO
							aReceiveBuffer[diReceiveCount]:= m_ReceiveBuffer[i];
							diReceiveCount:=(diReceiveCount+1) MOD SIZEOF(aReceiveBuffer);
						END_FOR

						m_ConnectionWatchdog(IN:=FALSE);(*reset connection watchdog*)
					END_CASE

				(*send data*)
				IF xStartSend	 THEN
					m_State := STATE_TX;
				END_IF

	STATE_TX:	 (* send TCP-message *)
		m_diReturn := SysSockSend(diSocket := m_Socket,
								  pbyBuffer := ADR(ptSendData^[m_count]),(*geändert V1.4 bisher: [0] *)
								  diBufferSize := diSendCount-m_count,
								  diFlags :=m_Flags);
		CASE m_diReturn OF
		-1:	(* ERROR or data could not yet be send (V1.3 due to new FW11) *)
			m_ConnectionWatchdog(IN:=TRUE , PT:=tServerTimeOut );
			IF m_connectionWatchdog.Q THEN
				m_State:= STATE_CLOSE;
				m_ConnectionWatchdog(IN:=FALSE);(*reset connection watchdog*)
				diError := 16#8007;
			END_IF
		0: (* socket was "gracefully closed"  *)
			m_State := STATE_CLOSE;
			diError := 16#8003;
		ELSE (* succesful *)
			m_count:=m_count+m_diReturn;
			IF m_count>=diSendCount THEN
				diError := 16#0000;
				m_State := STATE_RX;
				m_count:=0;
				xStartSend:=FALSE;
			END_IF
			m_ConnectionWatchdog(IN:=FALSE);(*reset connection watchdog*)
		END_CASE


		STATE_CLOSE:	(* Close the server *)

		IF ADR(%MW0)=16#30000000  OR ADR(%MW0)=16#20000000 THEN (*841 or 881*)
			;
		ELSE
			IF m_Socket>=0 THEN
				SysSockShutdown(m_Socket, 0);;(*870*)
			END_IF
		END_IF
		IF m_Socket>=0 THEN
			SysSockClose( m_Socket);
		END_IF
		xClientConnected:= FALSE;
		m_State:= STATE_OPEN; (* Try to open the server again *)
		m_ConnectionWatchdog(IN:=FALSE);(*reset connection watchdog*)

		STATE_ERROR_TRAP: (* Error Read/Write socket  *)
			m_State:= STATE_ERROR_TRAP;

	ELSE  (* Bad FSM code trap  *)
			m_State:= STATE_ERROR_TRAP;
			diError:= 16#8008;
	END_CASE;
ELSE
	IF m_State <> STATE_INIT THEN
		IF ADR(%MW0)=16#30000000  OR ADR(%MW0)=16#20000000 THEN (*841 or 881*)
			;
		ELSE
			IF m_Socket>=0 THEN
				SysSockShutdown(m_Socket, 0);;(*870*)
			END_IF
		END_IF
		IF m_Socket>=0 THEN
			SysSockClose( m_Socket);
		END_IF
		IF ADR(%MW0)=16#30000000  OR ADR(%MW0)=16#20000000 THEN (*841 or 881*)
			;
		ELSE
			IF m_ServerSocket>=0 THEN
				SysSockShutdown(m_ServerSocket, 0);;(*870*)
			END_IF
		END_IF
		IF m_ServerSocket>=0 THEN
			SysSockClose( m_ServerSocket);
		END_IF
		xClientConnected:= FALSE;
		diError:= 0;
		m_State:= STATE_init; (* Try to open the server again *)
		m_ConnectionWatchdog(IN:=FALSE);(*reset connection watchdog*)
	END_IF
END_IF
END_FUNCTION_BLOCK

(* POU Utils Functions/HEXTORAW, ST *)
FUNCTION HEXTORAW : WORD
VAR_INPUT
	pString		: POINTER TO BYTE;
	StringLen	: WORD;
	pData		: POINTER TO BYTE;
END_VAR
VAR
	xl: WORD;
	xi: WORD;
	xr: BYTE;
END_VAR
xl:=0;
xi:=0;

WHILE xi<StringLen DO

	IF pString^>=97 AND pString^<=102 THEN
		xr := pString^ - 87;
	ELSIF pString^>=65 AND pString^<=70 THEN
		xr := pString^ - 55;
	ELSIF pString^>=48 AND pString^<=57 THEN
		xr := pString^ - 48;
	ELSE
		xr := 16;
	END_IF

	IF xr<16 THEN
		IF (xi AND 1)=0 THEN
			pData^ := xr * 16;
		ELSE
			pData^ := pData^ + xr;
			pData := pData + 1;
			xl := xl + 1;
		END_IF
	END_IF

	xi := xi + 1;
	pString := pString + 1;

END_WHILE

HEXTORAW:=xl;
END_FUNCTION

(* POU Utils/USRLED_Update, ST *)
PROGRAM USRLED_Update
VAR
	OldStatus: en_SYS_Status;

	aFS : ARRAY [0..24] OF FLASHING_SEQUENCE :=
		(Colour:=GREEN,  Frequency:=1,   Relation:=128, Duration:=t#0s,    NextIndex:=0),  (* 0 => RUNNING *)
		(Colour:=ORANGE, Frequency:=1,   Relation:=128, Duration:=t#0s,    NextIndex:=1),  (* 1 => INIT *)
		(Colour:=RED,    Frequency:=4,   Relation:=128, Duration:=t#0s,    NextIndex:=2),  (* 2 => ERROR *)
		(Colour:=RED,    Frequency:=10,  Relation:=128, Duration:=t#0s,    NextIndex:=3),  (* 3 => ALARM *)
		(Colour:=ORANGE, Frequency:=200, Relation:=16,  Duration:=t#100ms, NextIndex:=11), (* 10 *)
		(Colour:=ORANGE, Frequency:=200, Relation:=32,  Duration:=t#100ms, NextIndex:=12),
		(Colour:=ORANGE, Frequency:=200, Relation:=64,  Duration:=t#100ms, NextIndex:=13),
		(Colour:=ORANGE, Frequency:=200, Relation:=128, Duration:=t#100ms, NextIndex:=14),
		(Colour:=ORANGE, Frequency:=200, Relation:=192, Duration:=t#100ms, NextIndex:=15),
		(Colour:=ORANGE, Frequency:=200, Relation:=128, Duration:=t#100ms, NextIndex:=16),
		(Colour:=ORANGE, Frequency:=200, Relation:=64,  Duration:=t#100ms, NextIndex:=17),
		(Colour:=ORANGE, Frequency:=200, Relation:=32,  Duration:=t#100ms, NextIndex:=18),
		(Colour:=ORANGE, Frequency:=200, Relation:=16,  Duration:=t#100ms, NextIndex:=19),
		(Colour:=ORANGE, Frequency:=200, Relation:=8,   Duration:=t#100ms, NextIndex:=10),
		(Colour:=GREEN,  Frequency:=200, Relation:=16,  Duration:=t#100ms, NextIndex:=21), (* 20 *)
		(Colour:=GREEN,  Frequency:=200, Relation:=32,  Duration:=t#100ms, NextIndex:=22),
		(Colour:=GREEN,  Frequency:=200, Relation:=64,  Duration:=t#100ms, NextIndex:=23),
		(Colour:=GREEN,  Frequency:=200, Relation:=128, Duration:=t#100ms, NextIndex:=24),
		(Colour:=GREEN,  Frequency:=200, Relation:=192, Duration:=t#100ms, NextIndex:=25),
		(Colour:=GREEN,  Frequency:=200, Relation:=128, Duration:=t#100ms, NextIndex:=26),
		(Colour:=GREEN,  Frequency:=200, Relation:=64,  Duration:=t#100ms, NextIndex:=27),
		(Colour:=GREEN,  Frequency:=200, Relation:=32,  Duration:=t#100ms, NextIndex:=28),
		(Colour:=GREEN,  Frequency:=200, Relation:=16,  Duration:=t#100ms, NextIndex:=29),
		(Colour:=GREEN,  Frequency:=200, Relation:=8,   Duration:=t#100ms, NextIndex:=20);

	pFS : POINTER TO FLASHING_SEQUENCE;


END_VAR
IF Sys.Status <> OldStatus THEN

	OldStatus:=Sys.Status;

	CASE OldStatus OF

		S_STARTUP:
			pFS:=ADR(aFS);
			SET_FLASHING_SEQUENCE(EN:=TRUE, POINTER_TO_POINTER_TO_ARRAY:=ADR(pFS));
			SET_FLASHING_SEQUENCE_INDEX(EN:=TRUE, IMMEDIATE:=FALSE, INDEX:=1);
			START_FLASHING_SEQUENCE(EN:=TRUE);

		S_RUNNING:
			SET_FLASHING_SEQUENCE_INDEX(EN:=TRUE, IMMEDIATE:=TRUE, INDEX:=0);

	END_CASE

END_IF
END_PROGRAM

(* POU Plant/SYS_Proc, ST *)
PROGRAM SYS_Proc
VAR
(*	fALARM_PB		:FLT_TAP;
	fALARM_TB		:FLT_TAP;
	fALARM_PM		:FLT_TAP; *)

(*	fGZB_ST			:FLT_TAP;  (* GATEWAY ZIGBEE *)*)
	fVPN_ST1		:FLT_TAP;  (* VPN CONNECT *)
	fVPN_ST2		:FLT_TAP;  (* VPN STATUS *)
(*	fKEY_CT_ST		:FLT_TAP;  (* DOOR1 *)*)
(*	fKEY_SCT_ST		:FLT_TAP;  (* DOOR2 *)*)
	fKEY_QE_ST		:FLT_TAP;  (* DOOR3 *)

	x: BOOL;
END_VAR
(*************** ISPESL *****************)
(*
fALARM_PB(IN:=ALARM_PB);
IF fALARM_PB.EVH THEN
	LogEv(EL_AlarmStop,EO_PBV,1,1,'Over_Pressure_Alarm');
END_IF

fALARM_TB(IN:=ALARM_TB);
IF fALARM_TB.EVH THEN
	LogEv(EL_AlarmStop,EO_TBV,1,1,'Over_Temperature_Alarm');
END_IF

fALARM_PM(IN:=ALARM_PM);
IF fALARM_PM.EVH THEN
	LogEv(EL_AlarmStop,EO_PMV,1,1,'Under_Pressure_Alarm');
END_IF
*)
(****************************************)
(*
(*### VPN Connection Check ###*)
fVPN_ST1(IN:=VPN_ST1);
IF fVPN_ST1.EVH THEN
	LogEv(EL_Log,EO_VPN,1,1,'CONNECT_ON');
END_IF
IF fVPN_ST1.EVL THEN
	LogEv(EL_Log,EO_VPN,1,2,'CONNECT_OFF');
END_IF
*)
(*
(*### VPN Status Check ###*)
fVPN_ST2(IN:=VPN_ST2);
IF fVPN_ST2.EVH THEN
	LogEv(EL_Log,EO_VPN,1,3,'STATUS_UP');
END_IF
IF fVPN_ST2.EVL THEN
	LogEv(EL_Wrn,EO_VPN,1,4,'STATUS_DOWN');
END_IF
*)
(*### DOOR01 Status Check ###*)(*
fKEY_CT_ST(IN:=KEY_CT_ST);
IF fKEY_CT_ST.EVH THEN
	LogEv(EL_Log,EO_DOOR,1,2,'Centrale_termica_Close');
END_IF
IF fKEY_CT_ST.EVL THEN
	LogEv(EL_Wrn,EO_DOOR,1,1,'Centrale_termica_Open');
END_IF
*)
(*### DOOR02 Status Check ###*)(*
fKEY_SCT_ST(IN:=KEY_SCT_ST);
IF fKEY_SCT_ST.EVH THEN
	LogEv(EL_Log,EO_DOOR,2,2,'Sottocentrale_termica_Close');
END_IF
IF fKEY_SCT_ST.EVL THEN
	LogEv(EL_Wrn,EO_DOOR,2,1,'Sottocentrale_termica_Open');
END_IF
*)
(*
(*### DOOR03 Status Check ###*)
fKEY_QE_ST(IN:=KEY_QE_ST);
IF fKEY_QE_ST.EVH THEN
	LogEv(EL_Log,EO_DOOR,3,2,'Quadro_Close');
END_IF
IF fKEY_QE_ST.EVL THEN
	LogEv(EL_Wrn,EO_DOOR,3,1,'Quadro_Open');
END_IF
*)
x:=1;
END_PROGRAM

(* POU Utils Functions/FLT_TAP, ST *)
FUNCTION_BLOCK FLT_TAP
VAR_INPUT
	IN		: BOOL;
	TAP		: BYTE:=4;
	INITEV	: BOOL:=TRUE;
END_VAR
VAR_OUTPUT
	OUT		: BOOL;
	EVH		: BOOL;
	EVL		: BOOL;
END_VAR
VAR
	init	: BOOL:=FALSE;
	cnt		: BYTE;
END_VAR
EVH:=FALSE;
EVL:=FALSE;

IF NOT init THEN
	init := TRUE;
	IF INITEV THEN
		OUT  := NOT IN;
		cnt  := TAP;
	ELSE
		OUT  := IN;
	END_IF
END_IF

IF OUT<>IN THEN
	cnt:=cnt+1;
	IF cnt>TAP THEN
		OUT:=IN;
		cnt:=0;
		IF OUT THEN EVH:=TRUE; ELSE EVL:=TRUE; END_IF
	END_IF
ELSE
	cnt:=0;
END_IF
END_FUNCTION_BLOCK

(* POU Configuration/MODBUS_CONFIGURATION, ST *)
PROGRAM MODBUS_CONFIGURATION
VAR                                
END_VAR                            
(*
   <?xml version="1.0" encoding="UTF-16" standalone="yes"?>
<network xml_structure_version="1">
	<generator_settings minRTUTaskCycleTimeMs="5" minEthaskCycleTimeMs="5" ethSlaveMultiplier="0.1" rtuInterfaceMultiplier="0.1" taskGeneration="false"/>
</network>
                              
*)                                 
;
END_PROGRAM

(* POU Utils Functions/AVERAGE_T, ST *)
FUNCTION_BLOCK AVERAGE_T
VAR_INPUT
	IN: 	INT;
END_VAR
VAR_OUTPUT
	HI:		INT;
	AVG:	INT;
	LOW:	INT;
	ERR:	BOOL;
END_VAR
VAR
	sum:	DINT;
	cnt:	WORD;
END_VAR
IF cnt>=65000 THEN
	ERR:=TRUE;
	Read();
	sum := sum - AVG;
	cnt := cnt + 1;
END_IF

sum := sum + IN;
cnt := cnt + 1;

IF IN<LOW THEN  LOW:=IN; END_IF
IF IN>HI  THEN HI :=IN; END_IF
END_FUNCTION_BLOCK
ACTION Read:
AVG := DINT_TO_INT(sum/cnt);
END_ACTION
ACTION Reset:
HI:=IN;
AVG:=IN;
LOW:=IN;
ERR:=FALSE;

sum:=IN;
cnt:=1;
END_ACTION

(* POU Utils/CSV_Log, ST *)
FUNCTION CSV_Log : BOOL
VAR_INPUT
END_VAR
VAR CONSTANT
	LogFileName:STRING:='S:\LOGS_ID1V3.CSV';
END_VAR
VAR
	s1 : STRING(180);
	hFile: 	DWORD;
END_VAR
(* Check file presence *)
hFile:=SysFileOpen(LogFileName,'r');
IF hFile=0 THEN
	(*** File not exist *** Create file and write header *)
	hFile:=SysFileOpen(LogFileName,'w');
	IF hFile<>0 THEN
		(* Write CSV header *)
		s1:='DATE-TIME;T-Amb;T-CAL01-SetP;T-CAL01-Send;T-CAL01-Ret;T-VRD01-Send;T-VRD02-Send;';
		SysFileWrite(hFile, ADR(s1), LEN(s1));
		s1:='T-CIR01-Amb;T-CIR04-Amb;T-CIR05-Amb;T-CIR07-Amb;T-VRD01-AvgSend;T-VRD02-AvgSend';
		SysFileWrite(hFile, ADR(s1), LEN(s1));
		SysFileWrite(hFile, ADR(Logger_CRLF), LEN(Logger_CRLF));
	END_IF
ELSE
	(*** File exist *** Close file and reopen in append mode *)
	SysFileClose(hFile);
	hFile:=SysFileOpen(LogFileName,'a');
END_IF

(* Log to file *)
IF hFile<>0 THEN
	(* Date stamp *)
	s1:=REPLACE( Sys.Time_LogString , ' ' , 1 , 11 );
	SysFileWrite(hFile, ADR(s1), LEN(s1));
	(* Log data *)
(*	s1:=CONCAT(';', REAL_TO_STRING(INT_TO_REAL(T_AMB)/10) ); *)
	s1:=CONCAT(';', REAL_TO_STRING(INT_TO_REAL(1)/10) );
	s1:=CONCAT(s1 , ';' );
	SysFileWrite(hFile, ADR(s1), LEN(s1));
	(* Add line CRLF and close *)
	SysFileWrite(hFile, ADR(Logger_CRLF), LEN(Logger_CRLF));
	SysFileClose(hFile);
END_IF
END_FUNCTION

(* POU IMI/FUN/DWORD_OF_WORD, ST *)
FUNCTION DWORD_OF_WORD : DWORD
VAR_INPUT
	W1 : WORD;
	W0 : WORD;
END_VAR


(*
version 1.0	18. jul. 2009
programmer 	hugo
tested by		tobias

this function creates a Dword from 2 individual Words

*)
DWORD_OF_WORD := SHL(WORD_TO_DWORD(W1),16) OR WORD_TO_DWORD(W0);


(* revision history

hm	18. jul. 2009	rev 1.0
	original version

*)
END_FUNCTION

(* POU Utils Functions/FLT_EVENT, ST *)
FUNCTION_BLOCK FLT_EVENT
VAR_INPUT
	IN		: BOOL;
	INITEV	: BOOL:=TRUE;
END_VAR
VAR_OUTPUT
	EVH		: BOOL;
	EVL		: BOOL;
END_VAR
VAR
	init	: BOOL:=FALSE;
	old		: BOOL;
END_VAR
EVH:=FALSE;
EVL:=FALSE;

IF NOT init THEN
	init:=TRUE;
	IF INITEV THEN
		old := NOT IN;
	ELSE
		old := IN;
	END_IF
END_IF

IF old<>IN THEN
	old:=IN;
	IF IN THEN EVH:=TRUE; ELSE EVL:=TRUE; END_IF
END_IF
END_FUNCTION_BLOCK

(* POU Utils Functions/LINEAR, ST *)
FUNCTION LINEAR : INT (* Linear interpolation *)
VAR_INPUT
	PuntoMinX:INT;
	PuntoMaxX:INT;
	ValIn : INT;
	PuntoMinY:REAL;
	PuntoMaxY:REAL;
	Decimali: BYTE;
END_VAR
VAR
	Gain: REAL;
	PuntoMinX_R	:REAL;
	PuntoMaxX_R	:REAL;
	Linearizzazione_R:REAL;
END_VAR
PuntoMinX_R:=INT_TO_REAL(PuntoMinX);
PuntoMaxX_R:=INT_TO_REAL(PuntoMaxX);

Gain:=(PuntoMaxX_R-PuntoMinX_R)/(PuntoMaxY-PuntoMinY);	(* Calcolo in guadagno per la linarizzazione *)
Linearizzazione_R:=PuntoMinx+(Gain*(ValIn-PuntoMinY));	(* Ottengo il valore linearizzato *)

LINEAR:=REAL_TO_INT(Linearizzazione_R*(EXPT(10, Decimali)));  (* Ottengo intero con i decimai voluti *)
END_FUNCTION

(* POU TCP_Logger/LogTrig, ST *)
FUNCTION LogTrig : BOOL
VAR
	s1 : STRING(260);
	i  : BYTE;
	j  : WORD;
	x: INT;
	k:INT;
	TPV07: BOOL;
	TPV01: BOOL;
END_VAR
(*---------------------------------------------------------------*)
(*---------------------------------------------------------------*)
Logger.TLen:=0;
(* Set GET header *)
ADDSTRING(ADR(Logger.TData), ADR(Logger_GETSTART), Logger.TLen);

(* Insert Header *)
s1:=INSERT('ID=&V=1&D=',DWORD_TO_STRING(Plant_SN),3);
s1:=CONCAT(s1,Sys.Time_LogString);
s1:=CONCAT(s1,'&S=');
IF Sys.Alarm THEN i:=2; ELSIF Sys.Warning THEN i:=1; ELSE i:=0; END_IF
s1:=CONCAT(s1,BYTE_TO_STRING(i));
ADDSTRING(ADR(Logger.TData), ADR(s1), Logger.TLen);

(* Insert PLC *)
s1:=CONCAT('&PLC=',INT_TO_STRING(Sistem_Status));
s1:=CONCAT(s1,';'); s1:=CONCAT(s1,INT_TO_STRING(BATTERY_STATUS));
s1:=CONCAT(s1,';'); s1:=CONCAT(s1,WORD_TO_STRING(SYSTEM_STATUS_COMMAND));
s1:=CONCAT(s1,';'); s1:=CONCAT(s1,WORD_TO_STRING(STATUS_DIGITAL_INPUT_1));
s1:=CONCAT(s1,';'); s1:=CONCAT(s1,WORD_TO_STRING(STATUS_DIGITAL_OUTPUT_1));
s1:=CONCAT(s1,';'); s1:=CONCAT(s1,WORD_TO_STRING(STATUS_SYSTEM_WARNNG_1));
s1:=CONCAT(s1,';'); s1:=CONCAT(s1,WORD_TO_STRING(STATUS_SYSTEM_ALARM_1));
s1:=CONCAT(s1,';'); s1:=CONCAT(s1,WORD_TO_STRING(STATUS_SYSTEM_ALARM_2));
s1:=CONCAT(s1,';'); s1:=CONCAT(s1,REAL_TO_STRING(PM1_Voltage_L12));
s1:=CONCAT(s1,';'); s1:=CONCAT(s1,REAL_TO_STRING(PM1_Voltage_L23));
s1:=CONCAT(s1,';'); s1:=CONCAT(s1,REAL_TO_STRING(PM1_Voltage_L31));
s1:=CONCAT(s1,';'); s1:=CONCAT(s1,REAL_TO_STRING(PM1_Current_L12));
s1:=CONCAT(s1,';'); s1:=CONCAT(s1,REAL_TO_STRING(PM1_Current_L23));
s1:=CONCAT(s1,';'); s1:=CONCAT(s1,REAL_TO_STRING(PM1_Current_L31));
s1:=CONCAT(s1,';'); s1:=CONCAT(s1,REAL_TO_STRING(PM1_Active_Power_Total));
s1:=CONCAT(s1,';'); s1:=CONCAT(s1,REAL_TO_STRING(PM1_Reactive_Power_Total));
s1:=CONCAT(s1,';'); s1:=CONCAT(s1,REAL_TO_STRING(PM1_Apparent_Power_Total));
s1:=CONCAT(s1,';'); s1:=CONCAT(s1,REAL_TO_STRING(PM1_Frequency));
s1:=CONCAT(s1,';'); s1:=CONCAT(s1,REAL_TO_STRING(PM1_Power_Factor_Total));
ADDSTRING(ADR(Logger.TData), ADR(s1), Logger.TLen);


(* Insert GATEWAY BATTERY *)
s1:=CONCAT('&GW=',REAL_TO_STRING(GW_Actual_DC_Voltage));
s1:=CONCAT(s1,';'); s1:=CONCAT(s1,REAL_TO_STRING(GW_Actual_DC_Current));
s1:=CONCAT(s1,';'); s1:=CONCAT(s1,REAL_TO_STRING(GW_Actual_Battery_SOC));
s1:=CONCAT(s1,';'); s1:=CONCAT(s1,REAL_TO_STRING(GW_Actual_Heaters_Current));
s1:=CONCAT(s1,';'); s1:=CONCAT(s1,REAL_TO_STRING(GW_Vdc_Link_Request));
s1:=CONCAT(s1,';'); s1:=CONCAT(s1,REAL_TO_STRING(GW_Limit_Discharge_Current));
s1:=CONCAT(s1,';'); s1:=CONCAT(s1,REAL_TO_STRING(GW_Limit_Charge_Current));
s1:=CONCAT(s1,';'); s1:=CONCAT(s1,REAL_TO_STRING(GW_Min_DC_Voltage));
s1:=CONCAT(s1,';'); s1:=CONCAT(s1,REAL_TO_STRING(GW_Max_DC_Voltage));
s1:=CONCAT(s1,';'); s1:=CONCAT(s1,REAL_TO_STRING(GW_Actual_Battery_Capacity));
s1:=CONCAT(s1,';'); s1:=CONCAT(s1,REAL_TO_STRING(GW_Max_Battery_Voltage));
s1:=CONCAT(s1,';'); s1:=CONCAT(s1,REAL_TO_STRING(GW_Min_Battery_Voltage));
s1:=CONCAT(s1,';'); s1:=CONCAT(s1,REAL_TO_STRING(GW_Max_Battery_Temperature));
s1:=CONCAT(s1,';'); s1:=CONCAT(s1,REAL_TO_STRING(GW_Min_Battery_Temperature));
s1:=CONCAT(s1,';'); s1:=CONCAT(s1,REAL_TO_STRING(GW_Actual_DC_Power));
s1:=CONCAT(s1,';'); s1:=CONCAT(s1,INT_TO_STRING(GW_HOURSOp_Time));
s1:=CONCAT(s1,';'); s1:=CONCAT(s1,INT_TO_STRING(GW_MINOp_Time));
s1:=CONCAT(s1,';'); s1:=CONCAT(s1,INT_TO_STRING(GW_Status_Warning_1));
s1:=CONCAT(s1,';'); s1:=CONCAT(s1,INT_TO_STRING(GW_Status_Warning_2));
s1:=CONCAT(s1,';'); s1:=CONCAT(s1,INT_TO_STRING(GW_Status_Alarm_1));
s1:=CONCAT(s1,';'); s1:=CONCAT(s1,INT_TO_STRING(GW_Status_Alarm_2));
s1:=CONCAT(s1,';'); s1:=CONCAT(s1,INT_TO_STRING(GW_Status_Warning_A));
s1:=CONCAT(s1,';'); s1:=CONCAT(s1,INT_TO_STRING(GW_Status_Warning_B));
s1:=CONCAT(s1,';'); s1:=CONCAT(s1,INT_TO_STRING(GW_Status_Alarm_A));
s1:=CONCAT(s1,';'); s1:=CONCAT(s1,WORD_TO_STRING(GW_CONTROLWORD));
s1:=CONCAT(s1,';'); s1:=CONCAT(s1,WORD_TO_STRING(GW_STATUSWORD));
ADDSTRING(ADR(Logger.TData), ADR(s1), Logger.TLen);



(* PCS HPP 35*)
s1:=CONCAT('&PCS=',REAL_TO_STRING(PCS_Actual_Current_R));
s1:=CONCAT(s1,';'); s1:=CONCAT(s1,REAL_TO_STRING(PCS_Actual_Current_S));
s1:=CONCAT(s1,';'); s1:=CONCAT(s1,REAL_TO_STRING(PCS_Actual_Current_T));
s1:=CONCAT(s1,';'); s1:=CONCAT(s1,REAL_TO_STRING(PCS_Actual_Voltage_RS));
s1:=CONCAT(s1,';'); s1:=CONCAT(s1,REAL_TO_STRING(PCS_Actual_Voltage_ST));
s1:=CONCAT(s1,';'); s1:=CONCAT(s1,REAL_TO_STRING(PCS_Actual_Voltage_TR));
s1:=CONCAT(s1,';'); s1:=CONCAT(s1,REAL_TO_STRING(PCS_Frequency));
s1:=CONCAT(s1,';'); s1:=CONCAT(s1,REAL_TO_STRING(PCS_P_Actual));
s1:=CONCAT(s1,';'); s1:=CONCAT(s1,REAL_TO_STRING(PCS_Q_Actual));
s1:=CONCAT(s1,';'); s1:=CONCAT(s1,REAL_TO_STRING(PCS_A_Actual));
s1:=CONCAT(s1,';'); s1:=CONCAT(s1,REAL_TO_STRING(PCS_Battery_Voltage));
s1:=CONCAT(s1,';'); s1:=CONCAT(s1,REAL_TO_STRING(PCS_Battery_Current));
s1:=CONCAT(s1,';'); s1:=CONCAT(s1,REAL_TO_STRING(PCS_Battery_Power));
s1:=CONCAT(s1,';'); s1:=CONCAT(s1,REAL_TO_STRING(PCS_PV_Voltage));
s1:=CONCAT(s1,';'); s1:=CONCAT(s1,REAL_TO_STRING(PCS_PV_Current));
s1:=CONCAT(s1,';'); s1:=CONCAT(s1,REAL_TO_STRING(PCS_PV_Power));
s1:=CONCAT(s1,';'); s1:=CONCAT(s1,INT_TO_STRING(PCS_HPP_Status));
s1:=CONCAT(s1,';'); s1:=CONCAT(s1,INT_TO_STRING(PCS_Drive_Status));
s1:=CONCAT(s1,';'); s1:=CONCAT(s1,INT_TO_STRING(PCS_Chopper_Status));
s1:=CONCAT(s1,';'); s1:=CONCAT(s1,INT_TO_STRING(PCS_Run_Mode));
s1:=CONCAT(s1,';'); s1:=CONCAT(s1,WORD_TO_STRING(PCS_Drive_Warning_1));
s1:=CONCAT(s1,';'); s1:=CONCAT(s1,WORD_TO_STRING(PCS_Drive_Alarm_1));
s1:=CONCAT(s1,';'); s1:=CONCAT(s1,WORD_TO_STRING(PCS_HPP_Warning_1));
s1:=CONCAT(s1,';'); s1:=CONCAT(s1,WORD_TO_STRING(PCS_HPP_Alarm_1));
ADDSTRING(ADR(Logger.TData), ADR(s1), Logger.TLen);



(* Finalize string *)
ADDSTRING(ADR(Logger.TData), ADR(Logger_GETEND), Logger.TLen);

(*---------------------------------------------------------------*)
(*---------------------------------------------------------------*)

Logger_Send();
END_FUNCTION

(* POU Utils Functions/MEMCLR, ST *)
FUNCTION MEMCLR:BOOL
VAR_INPUT
	pDestinationAddress:POINTER TO ARRAY[1..2] OF BYTE;
	BytesToClear:WORD;
END_VAR
VAR
END_VAR
WHILE (BytesToClear > 0) DO
	pDestinationAddress^[1]:=0;
	pDestinationAddress:=ADR(pDestinationAddress^[2]); (* increment destination *)
	BytesToClear:=BytesToClear -1; (* decrement number of bytes to copy *)
END_WHILE
END_FUNCTION

(* POU PLC_WDT, ST *)
FUNCTION PLC_WDT: DWORD VAR_INPUT dwEvent: DWORD; dwFilter: DWORD; dwOwner: DWORD; END_VAR
LogEv(EL_AlarmStop,EO_SYS,1,10,'Watchdog');
END_FUNCTION

(* POU Utils Functions/RAWTOHEX, ST *)
FUNCTION RAWTOHEX : WORD
VAR_INPUT
	pData: POINTER TO BYTE;
	DataLen: WORD;
	pString: POINTER TO BYTE;
END_VAR
VAR
	xl: WORD;
END_VAR
xl:=0;

WHILE DataLen>0 DO

	pString^ := (pData^ / 16#10) + 48 + (((pData^ / 16#10)/10)*7);
	pString:=pString+1;
	pString^ := (pData^ AND 16#0F)  + 48 + (((pData^ AND 16#0F)/10)*7);
	pString:=pString+1;
	pData:=pData+1;
	DataLen:=DataLen-1;
	xl:=xl+2;

END_WHILE

(*pString^:=0;*)

RAWTOHEX:=xl;
END_FUNCTION

(* POU Utils Functions/RAWTOHEXSTR, ST *)
FUNCTION RAWTOHEXSTR : STRING(128)
VAR_INPUT
	pData: POINTER TO BYTE;
	DataLen: BYTE;
END_VAR
VAR
	pt: POINTER TO BYTE;
	xl: BYTE;
END_VAR
pt:=ADR(RAWTOHEXSTR);

xl:=2;

WHILE DataLen>0 AND xl<128 DO

	pt^ := (pData^ / 16#10) + 48 + (((pData^ / 16#10)/10)*7);
	pt:=pt+1;
	pt^ := (pData^ AND 16#0F)  + 48 + (((pData^ AND 16#0F)/10)*7);
	pt:=pt+1;

	xl:=xl+2;

	DataLen:=DataLen-1;
	pData:=pData+1;

END_WHILE

pt^:=0;
END_FUNCTION

(* POU Utils/RTC_Update, ST *)
FUNCTION RTC_Update : BOOL
VAR
	T: DT;
	TS: STRING;
	TS2: STRING;
	Hour: BYTE;
	Minute: BYTE;
END_VAR
(* Get RTC time *)
T:=SysRtcGetTime(TRUE);
Sys.Time_CT_DT:=T;
(* Calculate variables *)
TS:=DT_TO_STRING(T);
Sys.Time_LogString:=DELETE(STR:=TS, LEN:=3, POS:=1);
TS2:=MID(STR:=TS, LEN:=4, POS:= 4); Sys.Time_Year 	:=STRING_TO_WORD(TS2);
TS2:=MID(STR:=TS, LEN:=2, POS:= 9); Sys.Time_Month	:=STRING_TO_BYTE(TS2);
TS2:=MID(STR:=TS, LEN:=2, POS:=12); Sys.Time_Day  	:=STRING_TO_BYTE(TS2);
Sys.Time_CT_Day:=(32*(Sys.Time_Month-1)+Sys.Time_Day-1);
TS2:=MID(STR:=TS, LEN:=2, POS:=15); Hour			:=STRING_TO_BYTE(TS2);
TS2:=MID(STR:=TS, LEN:=2, POS:=18); Minute		 	:=STRING_TO_BYTE(TS2);
Sys.Time_CT_Quarter:=Hour*4+(Minute/15);
END_FUNCTION

(* Visualisation PLC_VISU
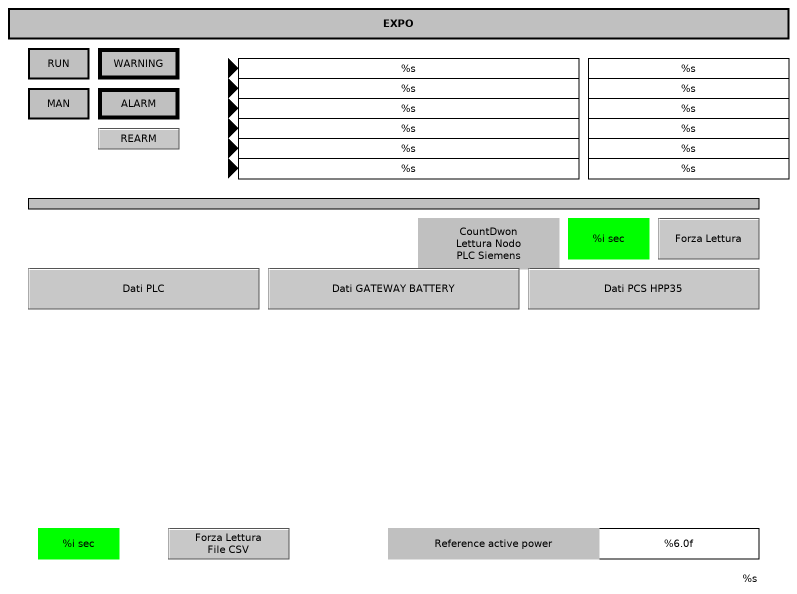
rectangle at (520,570)-(761,591): text "%s"; shows Sys.Time_LogString
rectangle at (10,10)-(791,41): text "EXPO"
rounded rectangle at (30,50)-(91,81): text "RUN"; alarm colour if NOT Mode_Manual; runs INTERN ASSIGN Mode_Manual:=(FALSE)
rounded rectangle at (30,90)-(91,121): text "MAN"; alarm colour if Mode_Manual; runs INTERN ASSIGN Mode_Manual:=(TRUE)
button at (30,270)-(261,311): text "Dati PLC"; opens WebVisu_PLC
rectangle at (590,60)-(791,81): text "%s"; shows Sys.LastLogs_Msg[0]
polygon at (230,160)-(240,180): invisible if Sys.LastLogs_Idx<>0
rectangle at (590,80)-(791,101): text "%s"; shows Sys.LastLogs_Msg[1]
polygon at (230,60)-(240,80): invisible if Sys.LastLogs_Idx<>1
rectangle at (590,100)-(791,121): text "%s"; shows Sys.LastLogs_Msg[2]
polygon at (230,80)-(240,100): invisible if Sys.LastLogs_Idx<>2
rectangle at (590,120)-(791,141): text "%s"; shows Sys.LastLogs_Msg[3]
polygon at (230,100)-(240,120): invisible if Sys.LastLogs_Idx<>3
rectangle at (590,140)-(791,161): text "%s"; shows Sys.LastLogs_Msg[4]
polygon at (230,120)-(240,140): invisible if Sys.LastLogs_Idx<>4
rectangle at (590,160)-(791,181): text "%s"; shows Sys.LastLogs_Msg[5]
polygon at (230,140)-(240,160): invisible if Sys.LastLogs_Idx<>5
rectangle at (240,60)-(581,81): text "%s"; shows Sys.LastLogs_Dat[0]
rectangle at (240,80)-(581,101): text "%s"; shows Sys.LastLogs_Dat[1]
rectangle at (240,100)-(581,121): text "%s"; shows Sys.LastLogs_Dat[2]
rectangle at (240,120)-(581,141): text "%s"; shows Sys.LastLogs_Dat[3]
rectangle at (240,140)-(581,161): text "%s"; shows Sys.LastLogs_Dat[4]
rectangle at (240,160)-(581,181): text "%s"; shows Sys.LastLogs_Dat[5]
rectangle at (100,90)-(181,121): text "ALARM"; alarm colour if Sys.Alarm; runs INTERN ASSIGN Mode_Manual:=(FALSE)
rectangle at (100,50)-(181,81): text "WARNING"; alarm colour if Sys.Warning; runs INTERN ASSIGN Mode_Manual:=(TRUE)
button at (100,130)-(181,151): text "REARM"; runs INTERN ASSIGN Sys.Alarm:=(FALSE);INTERN ASSIGN Sys.Warning:=(FALSE)
rectangle at (570,220)-(651,261): text "%i sec"; shows (TIME_TO_DINT(PLC_PRG.Timer2.PT)/1000)-(TIME_TO_DINT(PLC_PRG.Timer2.ET)/1000)
rectangle at (420,220)-(561,271): text "CountDwon / Lettura Nodo / PLC Siemens"
button at (660,220)-(761,261): text "Forza Lettura"; taps .ForzaLettura
rectangle at (600,530)-(761,561): text "%6.0f"; shows .Ref_P
rectangle at (390,530)-(601,561): text "Reference active power"
button at (270,270)-(521,311): text "Dati GATEWAY BATTERY"; opens WebVisu_GW
button at (530,270)-(761,311): text "Dati PCS HPP35"; opens WebVisu_PCS
rectangle at (40,530)-(121,561): text "%i sec"; shows (TIME_TO_DINT(PLC_PRG.Timer4.PT)/1000)-(TIME_TO_DINT(PLC_PRG.Timer4.ET)/1000)
button at (170,530)-(291,561): text "Forza Lettura / File CSV"; taps .ForzaLetturaCSV
1 more shapes without text or variables
3 elements of other kinds (tables, trends, ...) not read
*)

(* Visualisation WEBVISU_GW
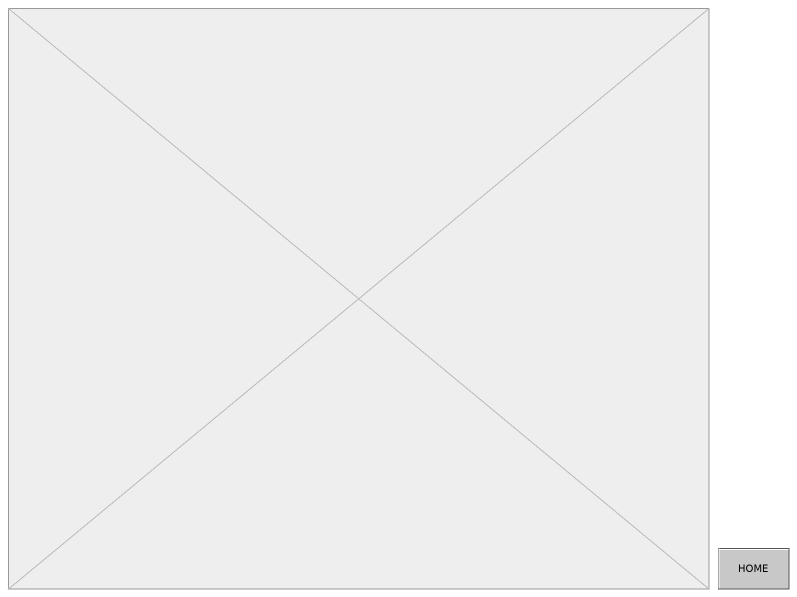
bitmap at (10,10)-(711,591): c:\users\esprinet 2014\documents\imi service\commesse\imi 15-438 expo\sviluppo\immagini\catturagw.jpg
button at (720,550)-(791,591): text "HOME"; opens PLC_Visu
26 elements of other kinds (tables, trends, ...) not read
*)

(* Visualisation WEBVISU_PCS
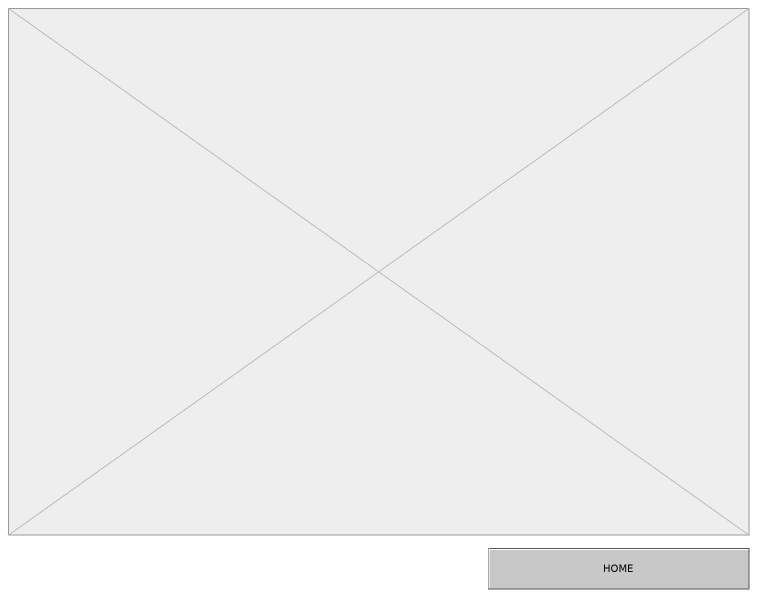
bitmap at (10,10)-(751,537): c:\users\esprinet 2014\documents\imi service\commesse\imi 15-438 expo\sviluppo\immagini\catturapcs.jpg
button at (490,550)-(751,591): text "HOME"; opens PLC_Visu
24 elements of other kinds (tables, trends, ...) not read
*)

(* Visualisation WEBVISU_PLC
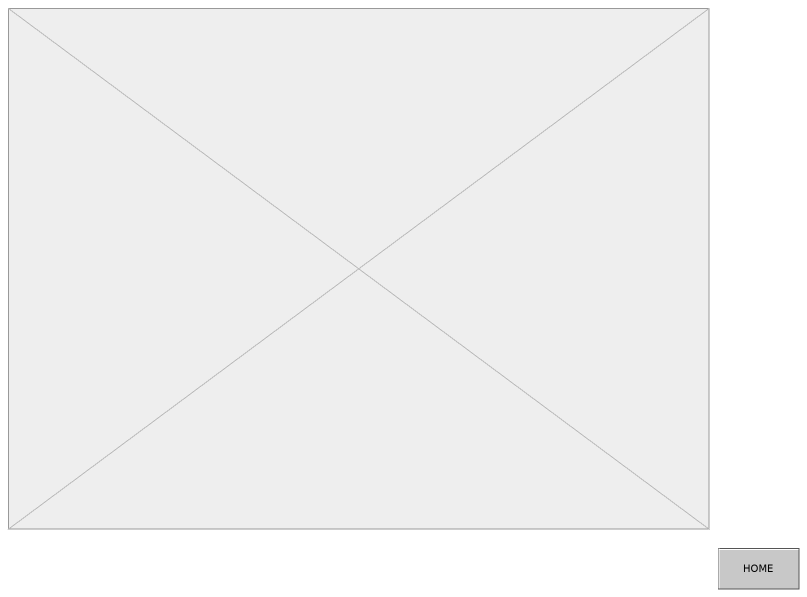
bitmap at (0,10)-(701,531): c:\users\esprinet 2014\documents\imi service\commesse\imi 15-438 expo\sviluppo\immagini\catturaplc.jpg
button at (710,550)-(791,591): text "HOME"; opens PLC_Visu
19 elements of other kinds (tables, trends, ...) not read
*)
